  gc_DbmTranslation_en_Text2282 : WSTRING(21) := "Variable debug Neotec";
  gc_DbmTranslation_en_Text2283 : WSTRING(21) := "Variable debug Neotec";
  gc_DbmTranslation_en_Text2284 : WSTRING(21) := "Variable debug Neotec";
  gc_DbmTranslation_en_Text2285 : WSTRING(21) := "Variable debug Neotec";
  gc_DbmTranslation_en_Text2286 : WSTRING(21) := "Variable debug Neotec";
  gc_DbmTranslation_en_Text2287 : WSTRING(21) := "Variable debug Neotec";
  gc_DbmTranslation_en_Text2288 : WSTRING(21) := "Variable debug Neotec";
  gc_DbmTranslation_en_Text2289 : WSTRING(21) := "Variable debug Neotec";
  gc_DbmTranslation_en_Text2290 : WSTRING(21) := "Variable debug Neotec";
  gc_DbmTranslation_en_Text2291 : WSTRING(21) := "Variable debug Neotec";
  gc_DbmTranslation_en_Text2292 : WSTRING(21) := "Variable debug Neotec";
  gc_DbmTranslation_en_Text2293 : WSTRING(21) := "Variable debug Neotec";
  gc_DbmTranslation_en_Text2294 : WSTRING(21) := "Variable debug Neotec";
  gc_DbmTranslation_en_Text2295 : WSTRING(21) := "Variable debug Neotec";
  gc_DbmTranslation_en_Text2296 : WSTRING(21) := "Variable debug Neotec";
  gc_DbmTranslation_en_Text2297 : WSTRING(21) := "Variable debug Neotec";
  gc_DbmTranslation_en_Text2298 : WSTRING(21) := "Variable debug Neotec";
  gc_DbmTranslation_en_Text2299 : WSTRING(21) := "Variable debug Neotec";
  gc_DbmTranslation_en_Text2300 : WSTRING(21) := "Variable debug Neotec";
  gc_DbmTranslation_en_Text2301 : WSTRING(21) := "Variable debug Neotec";
  gc_DbmTranslation_en_Text2302 : WSTRING(21) := "Variable debug Neotec";
  gc_DbmTranslation_en_Text2303 : WSTRING(21) := "Variable debug Neotec";
  gc_DbmTranslation_en_Text2304 : WSTRING(21) := "Variable debug Neotec";
  gc_DbmTranslation_en_Text2305 : WSTRING(21) := "Variable debug Neotec";
  gc_DbmTranslation_en_Text2306 : WSTRING(21) := "Variable debug Neotec";
  gc_DbmTranslation_en_Text2307 : WSTRING(21) := "Variable debug Neotec";
  gc_DbmTranslation_en_Text2308 : WSTRING(21) := "Variable debug Neotec";
  gc_DbmTranslation_en_Text2309 : WSTRING(21) := "Variable debug Neotec";
  gc_DbmTranslation_en_Text2310 : WSTRING(21) := "Variable debug Neotec";
  gc_DbmTranslation_en_Text2311 : WSTRING(64) := "Mesure de la température du liquide de refroidissement du moteur";
  gc_DbmTranslation_en_Text2312 : WSTRING(58) := "Pression mesuré dans le système de lubrification du moteur";
  gc_DbmTranslation_en_Text2313 : WSTRING(34) := "Vitesse actuelle du moteur calculé";
  gc_DbmTranslation_en_Text2314 : WSTRING(56) := "Courant de l'alternateur principale du moteur thermique ";
  gc_DbmTranslation_en_Text2315 : WSTRING(56) := "Etat du moteur : Motor stop, pre-start, Wram-Up,Starting";
  gc_DbmTranslation_en_Text2316 : WSTRING(40) := "Tension mesuré aux bornes de la batterie";
  gc_DbmTranslation_en_Text2317 : WSTRING(33) := "Commande de la vietesse du moteur";
  gc_DbmTranslation_en_Text2318 : WSTRING(30) := "Override Control Mode (SPN695)";
  gc_DbmTranslation_en_Text2319 : WSTRING(18) := "High pressure Oil ";
  gc_DbmTranslation_en_Text2320 : WSTRING(14) := "Warmin gActive";
  gc_DbmTranslation_en_Text2321 : WSTRING(10) := "Stop Motor";
  gc_DbmTranslation_en_Text2322 : WSTRING(27) := "Regeneration SOC at maximum";
  gc_DbmTranslation_en_Text2323 : WSTRING(61) := "Threshold maximum to autorize regeneration (Threshold of SOC)";
  gc_DbmTranslation_en_Text2324 : WSTRING(42) := "Hysteresis for regeneration of SOC maximum";
  gc_DbmTranslation_en_Text2325 : WSTRING(57) := "Number of time to refuse reloading from generator (Alarm)";
  gc_DbmTranslation_en_Text2326 : WSTRING(61) := "Number of time to refuse reloading from generator (forbidden)";
  gc_DbmTranslation_en_Text2327 : WSTRING(23) := "RPM motor maximum value";
  gc_DbmTranslation_en_Text2328 : WSTRING(23) := "RPM motor minimum value";
  gc_DbmTranslation_en_Text2329 : WSTRING(27) := "RPM for a movement with PVG";
  gc_DbmTranslation_en_Text2330 : WSTRING(27) := "RPM for a movement with TOR";
  gc_DbmTranslation_en_Text2331 : WSTRING(30) := "Hydraulic oil cold temperature";
  gc_DbmTranslation_en_Text2332 : WSTRING(42) := "Capacity of the battery in ampere per hour";
  gc_DbmTranslation_en_Text2333 : WSTRING(53) := "Number of element for the remaining regeneration time";
  gc_DbmTranslation_en_Text2334 : WSTRING(61) := "Number of times the alarm regeneration threshold was exceeded";
  gc_DbmTranslation_en_Text2335 : WSTRING(89) := "Number of times we exceeded the threshold of regeneration forbidden of the electric motor";
  gc_DbmTranslation_en_Text2336 : WSTRING(25) := "Cold Oil Tank Temperature";
  gc_DbmTranslation_en_Text2337 : WSTRING(30) := "Rpm Movements on Electric Mode";
  gc_DbmTranslation_en_Text2338 : WSTRING(37) := "Rpm Translation on Rail Electric Mode";
  gc_DbmTranslation_en_Text2339 : WSTRING(24) := "Rpm Oil Tank Temperature";
  gc_DbmTranslation_en_Text2340 : WSTRING(18) := "Rpm Electric motor";
  gc_DbmTranslation_en_Text2341 : WSTRING(12) := "Generator ON";
  gc_DbmTranslation_en_Text2342 : WSTRING(23) := "Automatic mode activate";
  gc_DbmTranslation_en_Text2343 : WSTRING(21) := "Silence mode activate";
  gc_DbmTranslation_en_Text2344 : WSTRING(21) := "Forcing mode activate";
  gc_DbmTranslation_en_Text2345 : WSTRING(24) := "Forcing regeneration Low";
  gc_DbmTranslation_en_Text2346 : WSTRING(25) := "Forcing regeneration High";
  gc_DbmTranslation_en_Text2347 : WSTRING(35) := "Remaining Regeneration time average";
  gc_DbmTranslation_en_Text2348 : WSTRING(25) := "Ask Reload With Generator";
  gc_DbmTranslation_en_Text2349 : WSTRING(27) := "Reloading With Generator On";
  gc_DbmTranslation_en_Text2350 : WSTRING(24) := "Stop regeneration by SOC";
  gc_DbmTranslation_en_Text2351 : WSTRING(24) := "Total regeneration Hours";
  gc_DbmTranslation_en_Text2352 : WSTRING(31) := "Picto Cold Oil Tank Temperature";
  gc_DbmTranslation_en_Text2353 : WSTRING(20) := "Total electric hours";
  gc_DbmTranslation_en_Text2354 : WSTRING(37) := "Picto recovery reduction ratio active";
  gc_DbVarGrpNameTranslation_en_Text2355 : WSTRING(17) := "NV_PARAMERTERS_C0";
  gc_DbVarGrpNameTranslation_en_Text2356 : WSTRING(23) := "NV_PARAM_SPEED_MAX_RAIL";
  gc_DbVarGrpNameTranslation_en_Text2357 : WSTRING(19) := "NV_PARAM_BRAKE_TEST";
  gc_DbVarGrpNameTranslation_en_Text2358 : WSTRING(28) := "NV_PARAM_RAIL_WORK_SAFETY_C0";
  gc_DbVarGrpNameTranslation_en_Text2359 : WSTRING(25) := "NV_PARAM_TRANSPORT_POS_C0";
  gc_DbVarGrpNameTranslation_en_Text2360 : WSTRING(28) := "NV_PARAM_SELECT_CONTROL_POST";
  gc_DbVarGrpNameTranslation_en_Text2361 : WSTRING(17) := "NV_PARAM_ALARM_C0";
  gc_DbVarGrpNameTranslation_en_Text2362 : WSTRING(21) := "NV_PARAM_MAST_DISPLAY";
  gc_DbVarGrpNameTranslation_en_Text2363 : WSTRING(17) := "NV_PARAMERTERS_C1";
  gc_DbVarGrpNameTranslation_en_Text2364 : WSTRING(17) := "NV_PARAM_MOTOR_C1";
  gc_DbVarGrpNameTranslation_en_Text2365 : WSTRING(31) := "NV_PARAM_LIMIT_WORK_ENVELOPE_C1";
  gc_DbVarGrpNameTranslation_en_Text2366 : WSTRING(24) := "NV_PARAM_MVT_END_STOP_C1";
  gc_DbVarGrpNameTranslation_en_Text2367 : WSTRING(21) := "NV_PARAM_AUTO_STOP_C1";
  gc_DbVarGrpNameTranslation_en_Text2368 : WSTRING(16) := "NV_PARAM_MAST_C1";
  gc_DbVarGrpNameTranslation_en_Text2369 : WSTRING(17) := "NV_PARAM_ALARM_C1";
  gc_DbVarGrpNameTranslation_en_Text2370 : WSTRING(12) := "NV_OPTION_C0";
  gc_DbVarGrpNameTranslation_en_Text2371 : WSTRING(12) := "NV_OPTION_C1";
  gc_DbmTranslation_en_Texts : ARRAY[0..2371] OF POINTER TO WSTRING(123) := [ADR(gc_DbmTranslation_en_Text0), ADR(gc_DbmTranslation_en_Text1), ADR(gc_DbmTranslation_en_Text2), ADR(gc_DbmTranslation_en_Text3), ADR(gc_DbmTranslation_en_Text4), ADR(gc_DbmTranslation_en_Text5), ADR(gc_DbmTranslation_en_Text6), ADR(gc_DbmTranslation_en_Text7), ADR(gc_DbmTranslation_en_Text8), ADR(gc_DbmTranslation_en_Text9), ADR(gc_DbmTranslation_en_Text10), ADR(gc_DbmTranslation_en_Text11), ADR(gc_DbmTranslation_en_Text12), ADR(gc_DbmTranslation_en_Text13), ADR(gc_DbmTranslation_en_Text14), ADR(gc_DbmTranslation_en_Text15), ADR(gc_DbmTranslation_en_Text16), ADR(gc_DbmTranslation_en_Text17), ADR(gc_DbmTranslation_en_Text18), ADR(gc_DbmTranslation_en_Text19), ADR(gc_DbmTranslation_en_Text20), ADR(gc_DbmTranslation_en_Text21), ADR(gc_DbmTranslation_en_Text22), ADR(gc_DbmTranslation_en_Text23), ADR(gc_DbmTranslation_en_Text24), ADR(gc_DbmTranslation_en_Text25), ADR(gc_DbmTranslation_en_Text26), ADR(gc_DbmTranslation_en_Text27), ADR(gc_DbmTranslation_en_Text28), ADR(gc_DbmTranslation_en_Text29), ADR(gc_DbmTranslation_en_Text30), ADR(gc_DbmTranslation_en_Text31), ADR(gc_DbmTranslation_en_Text32), ADR(gc_DbmTranslation_en_Text33), ADR(gc_DbmTranslation_en_Text34), ADR(gc_DbmTranslation_en_Text35), ADR(gc_DbmTranslation_en_Text36), ADR(gc_DbmTranslation_en_Text37), ADR(gc_DbmTranslation_en_Text38), ADR(gc_DbmTranslation_en_Text39), ADR(gc_DbmTranslation_en_Text40), ADR(gc_DbmTranslation_en_Text41), ADR(gc_DbmTranslation_en_Text42), ADR(gc_DbmTranslation_en_Text43), ADR(gc_DbmTranslation_en_Text44), ADR(gc_DbmTranslation_en_Text45), ADR(gc_DbmTranslation_en_Text46), ADR(gc_DbmTranslation_en_Text47), ADR(gc_DbmTranslation_en_Text48), ADR(gc_DbmTranslation_en_Text49), ADR(gc_DbmTranslation_en_Text50), ADR(gc_DbmTranslation_en_Text51), ADR(gc_DbmTranslation_en_Text52), ADR(gc_DbmTranslation_en_Text53), ADR(gc_DbmTranslation_en_Text54), ADR(gc_DbmTranslation_en_Text55), ADR(gc_DbmTranslation_en_Text56), ADR(gc_DbmTranslation_en_Text57), ADR(gc_DbmTranslation_en_Text58), ADR(gc_DbmTranslation_en_Text59), ADR(gc_DbmTranslation_en_Text60), ADR(gc_DbmTranslation_en_Text61), ADR(gc_DbmTranslation_en_Text62), ADR(gc_DbmTranslation_en_Text63), ADR(gc_DbmTranslation_en_Text64), ADR(gc_DbmTranslation_en_Text65), ADR(gc_DbmTranslation_en_Text66), ADR(gc_DbmTranslation_en_Text67), ADR(gc_DbmTranslation_en_Text68), ADR(gc_DbmTranslation_en_Text69), ADR(gc_DbmTranslation_en_Text70), ADR(gc_DbmTranslation_en_Text71), ADR(gc_DbmTranslation_en_Text72), ADR(gc_DbmTranslation_en_Text73), ADR(gc_DbmTranslation_en_Text74), ADR(gc_DbmTranslation_en_Text75), ADR(gc_DbmTranslation_en_Text76), ADR(gc_DbmTranslation_en_Text77), ADR(gc_DbmTranslation_en_Text78), ADR(gc_DbmTranslation_en_Text79), ADR(gc_DbmTranslation_en_Text80), ADR(gc_DbmTranslation_en_Text81), ADR(gc_DbmTranslation_en_Text82), ADR(gc_DbmTranslation_en_Text83), ADR(gc_DbmTranslation_en_Text84), ADR(gc_DbmTranslation_en_Text85), ADR(gc_DbmTranslation_en_Text86), ADR(gc_DbmTranslation_en_Text87), ADR(gc_DbmTranslation_en_Text88), ADR(gc_DbmTranslation_en_Text89), ADR(gc_DbmTranslation_en_Text90), ADR(gc_DbmTranslation_en_Text91), ADR(gc_DbmTranslation_en_Text92), ADR(gc_DbmTranslation_en_Text93), ADR(gc_DbmTranslation_en_Text94), ADR(gc_DbmTranslation_en_Text95), ADR(gc_DbmTranslation_en_Text96), ADR(gc_DbmTranslation_en_Text97), ADR(gc_DbmTranslation_en_Text98), ADR(gc_DbmTranslation_en_Text99), ADR(gc_DbmTranslation_en_Text100), ADR(gc_DbmTranslation_en_Text101), ADR(gc_DbmTranslation_en_Text102), ADR(gc_DbmTranslation_en_Text103), ADR(gc_DbmTranslation_en_Text104), ADR(gc_DbmTranslation_en_Text105), ADR(gc_DbmTranslation_en_Text106), ADR(gc_DbmTranslation_en_Text107), ADR(gc_DbmTranslation_en_Text108), ADR(gc_DbmTranslation_en_Text109), ADR(gc_DbmTranslation_en_Text110), ADR(gc_DbmTranslation_en_Text111), ADR(gc_DbmTranslation_en_Text112), ADR(gc_DbmTranslation_en_Text113), ADR(gc_DbmTranslation_en_Text114), ADR(gc_DbmTranslation_en_Text115), ADR(gc_DbmTranslation_en_Text116), ADR(gc_DbmTranslation_en_Text117), ADR(gc_DbmTranslation_en_Text118), ADR(gc_DbmTranslation_en_Text119), ADR(gc_DbmTranslation_en_Text120), ADR(gc_DbmTranslation_en_Text121), ADR(gc_DbmTranslation_en_Text122), ADR(gc_DbmTranslation_en_Text123), ADR(gc_DbmTranslation_en_Text124), ADR(gc_DbmTranslation_en_Text125), ADR(gc_DbmTranslation_en_Text126), ADR(gc_DbmTranslation_en_Text127), ADR(gc_DbmTranslation_en_Text128), ADR(gc_DbmTranslation_en_Text129), ADR(gc_DbmTranslation_en_Text130), ADR(gc_DbmTranslation_en_Text131), ADR(gc_DbmTranslation_en_Text132), ADR(gc_DbmTranslation_en_Text133), ADR(gc_DbmTranslation_en_Text134), ADR(gc_DbmTranslation_en_Text135), ADR(gc_DbmTranslation_en_Text136), ADR(gc_DbmTranslation_en_Text137), ADR(gc_DbmTranslation_en_Text138), ADR(gc_DbmTranslation_en_Text139), ADR(gc_DbmTranslation_en_Text140), ADR(gc_DbmTranslation_en_Text141), ADR(gc_DbmTranslation_en_Text142), ADR(gc_DbmTranslation_en_Text143), ADR(gc_DbmTranslation_en_Text144), ADR(gc_DbmTranslation_en_Text145), ADR(gc_DbmTranslation_en_Text146), ADR(gc_DbmTranslation_en_Text147), ADR(gc_DbmTranslation_en_Text148), ADR(gc_DbmTranslation_en_Text149), ADR(gc_DbmTranslation_en_Text150), ADR(gc_DbmTranslation_en_Text151), ADR(gc_DbmTranslation_en_Text152), ADR(gc_DbmTranslation_en_Text153), ADR(gc_DbmTranslation_en_Text154), ADR(gc_DbmTranslation_en_Text155), ADR(gc_DbmTranslation_en_Text156), ADR(gc_DbmTranslation_en_Text157), ADR(gc_DbmTranslation_en_Text158), ADR(gc_DbmTranslation_en_Text159), ADR(gc_DbmTranslation_en_Text160), ADR(gc_DbmTranslation_en_Text161), ADR(gc_DbmTranslation_en_Text162), ADR(gc_DbmTranslation_en_Text163), ADR(gc_DbmTranslation_en_Text164), ADR(gc_DbmTranslation_en_Text165), ADR(gc_DbmTranslation_en_Text166), ADR(gc_DbmTranslation_en_Text167), ADR(gc_DbmTranslation_en_Text168), ADR(gc_DbmTranslation_en_Text169), ADR(gc_DbmTranslation_en_Text170), ADR(gc_DbmTranslation_en_Text171), ADR(gc_DbmTranslation_en_Text172), ADR(gc_DbmTranslation_en_Text173), ADR(gc_DbmTranslation_en_Text174), ADR(gc_DbmTranslation_en_Text175), ADR(gc_DbmTranslation_en_Text176), ADR(gc_DbmTranslation_en_Text177), ADR(gc_DbmTranslation_en_Text178), ADR(gc_DbmTranslation_en_Text179), ADR(gc_DbmTranslation_en_Text180), ADR(gc_DbmTranslation_en_Text181), ADR(gc_DbmTranslation_en_Text182), ADR(gc_DbmTranslation_en_Text183), ADR(gc_DbmTranslation_en_Text184), ADR(gc_DbmTranslation_en_Text185), ADR(gc_DbmTranslation_en_Text186), ADR(gc_DbmTranslation_en_Text187), ADR(gc_DbmTranslation_en_Text188), ADR(gc_DbmTranslation_en_Text189), ADR(gc_DbmTranslation_en_Text190), ADR(gc_DbmTranslation_en_Text191), ADR(gc_DbmTranslation_en_Text192), ADR(gc_DbmTranslation_en_Text193), ADR(gc_DbmTranslation_en_Text194), ADR(gc_DbmTranslation_en_Text195), ADR(gc_DbmTranslation_en_Text196), ADR(gc_DbmTranslation_en_Text197), ADR(gc_DbmTranslation_en_Text198), ADR(gc_DbmTranslation_en_Text199), ADR(gc_DbmTranslation_en_Text200), ADR(gc_DbmTranslation_en_Text201), ADR(gc_DbmTranslation_en_Text202), ADR(gc_DbmTranslation_en_Text203), ADR(gc_DbmTranslation_en_Text204), ADR(gc_DbmTranslation_en_Text205), ADR(gc_DbmTranslation_en_Text206), ADR(gc_DbmTranslation_en_Text207), ADR(gc_DbmTranslation_en_Text208), ADR(gc_DbmTranslation_en_Text209), ADR(gc_DbmTranslation_en_Text210), ADR(gc_DbmTranslation_en_Text211), ADR(gc_DbmTranslation_en_Text212), ADR(gc_DbmTranslation_en_Text213), ADR(gc_DbmTranslation_en_Text214), ADR(gc_DbmTranslation_en_Text215), ADR(gc_DbmTranslation_en_Text216), ADR(gc_DbmTranslation_en_Text217), ADR(gc_DbmTranslation_en_Text218), ADR(gc_DbmTranslation_en_Text219), ADR(gc_DbmTranslation_en_Text220), ADR(gc_DbmTranslation_en_Text221), ADR(gc_DbmTranslation_en_Text222), ADR(gc_DbmTranslation_en_Text223), ADR(gc_DbmTranslation_en_Text224), ADR(gc_DbmTranslation_en_Text225), ADR(gc_DbmTranslation_en_Text226), ADR(gc_DbmTranslation_en_Text227), ADR(gc_DbmTranslation_en_Text228), ADR(gc_DbmTranslation_en_Text229), ADR(gc_DbmTranslation_en_Text230), ADR(gc_DbmTranslation_en_Text231), ADR(gc_DbmTranslation_en_Text232), ADR(gc_DbmTranslation_en_Text233), ADR(gc_DbmTranslation_en_Text234), ADR(gc_DbmTranslation_en_Text235), ADR(gc_DbmTranslation_en_Text236), ADR(gc_DbmTranslation_en_Text237), ADR(gc_DbmTranslation_en_Text238), ADR(gc_DbmTranslation_en_Text239), ADR(gc_DbmTranslation_en_Text240), ADR(gc_DbmTranslation_en_Text241), ADR(gc_DbmTranslation_en_Text242), ADR(gc_DbmTranslation_en_Text243), ADR(gc_DbmTranslation_en_Text244), ADR(gc_DbmTranslation_en_Text245), ADR(gc_DbmTranslation_en_Text246), ADR(gc_DbmTranslation_en_Text247), ADR(gc_DbmTranslation_en_Text248), ADR(gc_DbmTranslation_en_Text249), ADR(gc_DbmTranslation_en_Text250), ADR(gc_DbmTranslation_en_Text251), ADR(gc_DbmTranslation_en_Text252), ADR(gc_DbmTranslation_en_Text253), ADR(gc_DbmTranslation_en_Text254), ADR(gc_DbmTranslation_en_Text255), ADR(gc_DbmTranslation_en_Text256), ADR(gc_DbmTranslation_en_Text257), ADR(gc_DbmTranslation_en_Text258), ADR(gc_DbmTranslation_en_Text259), ADR(gc_DbmTranslation_en_Text260), ADR(gc_DbmTranslation_en_Text261), ADR(gc_DbmTranslation_en_Text262), ADR(gc_DbmTranslation_en_Text263), ADR(gc_DbmTranslation_en_Text264), ADR(gc_DbmTranslation_en_Text265), ADR(gc_DbmTranslation_en_Text266), ADR(gc_DbmTranslation_en_Text267), ADR(gc_DbmTranslation_en_Text268), ADR(gc_DbmTranslation_en_Text269), ADR(gc_DbmTranslation_en_Text270), ADR(gc_DbmTranslation_en_Text271), ADR(gc_DbmTranslation_en_Text272), ADR(gc_DbmTranslation_en_Text273), ADR(gc_DbmTranslation_en_Text274), ADR(gc_DbmTranslation_en_Text275), ADR(gc_DbmTranslation_en_Text276), ADR(gc_DbmTranslation_en_Text277), ADR(gc_DbmTranslation_en_Text278), ADR(gc_DbmTranslation_en_Text279), ADR(gc_DbmTranslation_en_Text280), ADR(gc_DbmTranslation_en_Text281), ADR(gc_DbmTranslation_en_Text282), ADR(gc_DbmTranslation_en_Text283), ADR(gc_DbmTranslation_en_Text284), ADR(gc_DbmTranslation_en_Text285), ADR(gc_DbmTranslation_en_Text286), ADR(gc_DbmTranslation_en_Text287), ADR(gc_DbmTranslation_en_Text288), ADR(gc_DbmTranslation_en_Text289), ADR(gc_DbmTranslation_en_Text290), ADR(gc_DbmTranslation_en_Text291), ADR(gc_DbmTranslation_en_Text292), ADR(gc_DbmTranslation_en_Text293), ADR(gc_DbmTranslation_en_Text294), ADR(gc_DbmTranslation_en_Text295), ADR(gc_DbmTranslation_en_Text296), ADR(gc_DbmTranslation_en_Text297), ADR(gc_DbmTranslation_en_Text298), ADR(gc_DbmTranslation_en_Text299), ADR(gc_DbmTranslation_en_Text300), ADR(gc_DbmTranslation_en_Text301), ADR(gc_DbmTranslation_en_Text302), ADR(gc_DbmTranslation_en_Text303), ADR(gc_DbmTranslation_en_Text304), ADR(gc_DbmTranslation_en_Text305), ADR(gc_DbmTranslation_en_Text306), ADR(gc_DbmTranslation_en_Text307), ADR(gc_DbmTranslation_en_Text308), ADR(gc_DbmTranslation_en_Text309), ADR(gc_DbmTranslation_en_Text310), ADR(gc_DbmTranslation_en_Text311), ADR(gc_DbmTranslation_en_Text312), ADR(gc_DbmTranslation_en_Text313), ADR(gc_DbmTranslation_en_Text314), ADR(gc_DbmTranslation_en_Text315), ADR(gc_DbmTranslation_en_Text316), ADR(gc_DbmTranslation_en_Text317), ADR(gc_DbmTranslation_en_Text318), ADR(gc_DbmTranslation_en_Text319), ADR(gc_DbmTranslation_en_Text320), ADR(gc_DbmTranslation_en_Text321), ADR(gc_DbmTranslation_en_Text322), ADR(gc_DbmTranslation_en_Text323), ADR(gc_DbmTranslation_en_Text324), ADR(gc_DbmTranslation_en_Text325), ADR(gc_DbmTranslation_en_Text326), ADR(gc_DbmTranslation_en_Text327), ADR(gc_DbmTranslation_en_Text328), ADR(gc_DbmTranslation_en_Text329), ADR(gc_DbmTranslation_en_Text330), ADR(gc_DbmTranslation_en_Text331), ADR(gc_DbmTranslation_en_Text332), ADR(gc_DbmTranslation_en_Text333), ADR(gc_DbmTranslation_en_Text334), ADR(gc_DbmTranslation_en_Text335), ADR(gc_DbmTranslation_en_Text336), ADR(gc_DbmTranslation_en_Text337), ADR(gc_DbmTranslation_en_Text338), ADR(gc_DbmTranslation_en_Text339), ADR(gc_DbmTranslation_en_Text340), ADR(gc_DbmTranslation_en_Text341), ADR(gc_DbmTranslation_en_Text342), ADR(gc_DbmTranslation_en_Text343), ADR(gc_DbmTranslation_en_Text344), ADR(gc_DbmTranslation_en_Text345), ADR(gc_DbmTranslation_en_Text346), ADR(gc_DbmTranslation_en_Text347), ADR(gc_DbmTranslation_en_Text348), ADR(gc_DbmTranslation_en_Text349), ADR(gc_DbmTranslation_en_Text350), ADR(gc_DbmTranslation_en_Text351), ADR(gc_DbmTranslation_en_Text352), ADR(gc_DbmTranslation_en_Text353), ADR(gc_DbmTranslation_en_Text354), ADR(gc_DbmTranslation_en_Text355), ADR(gc_DbmTranslation_en_Text356), ADR(gc_DbmTranslation_en_Text357), ADR(gc_DbmTranslation_en_Text358), ADR(gc_DbmTranslation_en_Text359), ADR(gc_DbmTranslation_en_Text360), ADR(gc_DbmTranslation_en_Text361), ADR(gc_DbmTranslation_en_Text362), ADR(gc_DbmTranslation_en_Text363), ADR(gc_DbmTranslation_en_Text364), ADR(gc_DbmTranslation_en_Text365), ADR(gc_DbmTranslation_en_Text366), ADR(gc_DbmTranslation_en_Text367), ADR(gc_DbmTranslation_en_Text368), ADR(gc_DbmTranslation_en_Text369), ADR(gc_DbmTranslation_en_Text370), ADR(gc_DbmTranslation_en_Text371), ADR(gc_DbmTranslation_en_Text372), ADR(gc_DbmTranslation_en_Text373), ADR(gc_DbmTranslation_en_Text374), ADR(gc_DbmTranslation_en_Text375), ADR(gc_DbmTranslation_en_Text376), ADR(gc_DbmTranslation_en_Text377), ADR(gc_DbmTranslation_en_Text378), ADR(gc_DbmTranslation_en_Text379), ADR(gc_DbmTranslation_en_Text380), ADR(gc_DbmTranslation_en_Text381), ADR(gc_DbmTranslation_en_Text382), ADR(gc_DbmTranslation_en_Text383), ADR(gc_DbmTranslation_en_Text384), ADR(gc_DbmTranslation_en_Text385), ADR(gc_DbmTranslation_en_Text386), ADR(gc_DbmTranslation_en_Text387), ADR(gc_DbmTranslation_en_Text388), ADR(gc_DbmTranslation_en_Text389), ADR(gc_DbmTranslation_en_Text390), ADR(gc_DbmTranslation_en_Text391), ADR(gc_DbmTranslation_en_Text392), ADR(gc_DbmTranslation_en_Text393), ADR(gc_DbmTranslation_en_Text394), ADR(gc_DbmTranslation_en_Text395), ADR(gc_DbmTranslation_en_Text396), ADR(gc_DbmTranslation_en_Text397), ADR(gc_DbmTranslation_en_Text398), ADR(gc_DbmTranslation_en_Text399), ADR(gc_DbmTranslation_en_Text400), ADR(gc_DbmTranslation_en_Text401), ADR(gc_DbmTranslation_en_Text402), ADR(gc_DbmTranslation_en_Text403), ADR(gc_DbmTranslation_en_Text404), ADR(gc_DbmTranslation_en_Text405), ADR(gc_DbmTranslation_en_Text406), ADR(gc_DbmTranslation_en_Text407), ADR(gc_DbmTranslation_en_Text408), ADR(gc_DbmTranslation_en_Text409), ADR(gc_DbmTranslation_en_Text410), ADR(gc_DbmTranslation_en_Text411), ADR(gc_DbmTranslation_en_Text412), ADR(gc_DbmTranslation_en_Text413), ADR(gc_DbmTranslation_en_Text414), ADR(gc_DbmTranslation_en_Text415), ADR(gc_DbmTranslation_en_Text416), ADR(gc_DbmTranslation_en_Text417), ADR(gc_DbmTranslation_en_Text418), ADR(gc_DbmTranslation_en_Text419), ADR(gc_DbmTranslation_en_Text420), ADR(gc_DbmTranslation_en_Text421), ADR(gc_DbmTranslation_en_Text422), ADR(gc_DbmTranslation_en_Text423), ADR(gc_DbmTranslation_en_Text424), ADR(gc_DbmTranslation_en_Text425), ADR(gc_DbmTranslation_en_Text426), ADR(gc_DbmTranslation_en_Text427), ADR(gc_DbmTranslation_en_Text428), ADR(gc_DbmTranslation_en_Text429), ADR(gc_DbmTranslation_en_Text430), ADR(gc_DbmTranslation_en_Text431), ADR(gc_DbmTranslation_en_Text432), ADR(gc_DbmTranslation_en_Text433), ADR(gc_DbmTranslation_en_Text434), ADR(gc_DbmTranslation_en_Text435), ADR(gc_DbmTranslation_en_Text436), ADR(gc_DbmTranslation_en_Text437), ADR(gc_DbmTranslation_en_Text438), ADR(gc_DbmTranslation_en_Text439), ADR(gc_DbmTranslation_en_Text440), ADR(gc_DbmTranslation_en_Text441), ADR(gc_DbmTranslation_en_Text442), ADR(gc_DbmTranslation_en_Text443), ADR(gc_DbmTranslation_en_Text444), ADR(gc_DbmTranslation_en_Text445), ADR(gc_DbmTranslation_en_Text446), ADR(gc_DbmTranslation_en_Text447), ADR(gc_DbmTranslation_en_Text448), ADR(gc_DbmTranslation_en_Text449), ADR(gc_DbmTranslation_en_Text450), ADR(gc_DbmTranslation_en_Text451), ADR(gc_DbmTranslation_en_Text452), ADR(gc_DbmTranslation_en_Text453), ADR(gc_DbmTranslation_en_Text454), ADR(gc_DbmTranslation_en_Text455), ADR(gc_DbmTranslation_en_Text456), ADR(gc_DbmTranslation_en_Text457), ADR(gc_DbmTranslation_en_Text458), ADR(gc_DbmTranslation_en_Text459), ADR(gc_DbmTranslation_en_Text460), ADR(gc_DbmTranslation_en_Text461), ADR(gc_DbmTranslation_en_Text462), ADR(gc_DbmTranslation_en_Text463), ADR(gc_DbmTranslation_en_Text464), ADR(gc_DbmTranslation_en_Text465), ADR(gc_DbmTranslation_en_Text466), ADR(gc_DbmTranslation_en_Text467), ADR(gc_DbmTranslation_en_Text468), ADR(gc_DbmTranslation_en_Text469), ADR(gc_DbmTranslation_en_Text470), ADR(gc_DbmTranslation_en_Text471), ADR(gc_DbmTranslation_en_Text472), ADR(gc_DbmTranslation_en_Text473), ADR(gc_DbmTranslation_en_Text474), ADR(gc_DbmTranslation_en_Text475), ADR(gc_DbmTranslation_en_Text476), ADR(gc_DbmTranslation_en_Text477), ADR(gc_DbmTranslation_en_Text478), ADR(gc_DbmTranslation_en_Text479), ADR(gc_DbmTranslation_en_Text480), ADR(gc_DbmTranslation_en_Text481), ADR(gc_DbmTranslation_en_Text482), ADR(gc_DbmTranslation_en_Text483), ADR(gc_DbmTranslation_en_Text484), ADR(gc_DbmTranslation_en_Text485), ADR(gc_DbmTranslation_en_Text486), ADR(gc_DbmTranslation_en_Text487), ADR(gc_DbmTranslation_en_Text488), ADR(gc_DbmTranslation_en_Text489), ADR(gc_DbmTranslation_en_Text490), ADR(gc_DbmTranslation_en_Text491), ADR(gc_DbmTranslation_en_Text492), ADR(gc_DbmTranslation_en_Text493), ADR(gc_DbmTranslation_en_Text494), ADR(gc_DbmTranslation_en_Text495), ADR(gc_DbmTranslation_en_Text496), ADR(gc_DbmTranslation_en_Text497), ADR(gc_DbmTranslation_en_Text498), ADR(gc_DbmTranslation_en_Text499), ADR(gc_DbmTranslation_en_Text500), ADR(gc_DbmTranslation_en_Text501), ADR(gc_DbmTranslation_en_Text502), ADR(gc_DbmTranslation_en_Text503), ADR(gc_DbmTranslation_en_Text504), ADR(gc_DbmTranslation_en_Text505), ADR(gc_DbmTranslation_en_Text506), ADR(gc_DbmTranslation_en_Text507), ADR(gc_DbmTranslation_en_Text508), ADR(gc_DbmTranslation_en_Text509), ADR(gc_DbmTranslation_en_Text510), ADR(gc_DbmTranslation_en_Text511), ADR(gc_DbmTranslation_en_Text512), ADR(gc_DbmTranslation_en_Text513), ADR(gc_DbmTranslation_en_Text514), ADR(gc_DbmTranslation_en_Text515), ADR(gc_DbmTranslation_en_Text516), ADR(gc_DbmTranslation_en_Text517), ADR(gc_DbmTranslation_en_Text518), ADR(gc_DbmTranslation_en_Text519), ADR(gc_DbmTranslation_en_Text520), ADR(gc_DbmTranslation_en_Text521), ADR(gc_DbmTranslation_en_Text522), ADR(gc_DbmTranslation_en_Text523), ADR(gc_DbmTranslation_en_Text524), ADR(gc_DbmTranslation_en_Text525), ADR(gc_DbmTranslation_en_Text526), ADR(gc_DbmTranslation_en_Text527), ADR(gc_DbmTranslation_en_Text528), ADR(gc_DbmTranslation_en_Text529), ADR(gc_DbmTranslation_en_Text530), ADR(gc_DbmTranslation_en_Text531), ADR(gc_DbmTranslation_en_Text532), ADR(gc_DbmTranslation_en_Text533), ADR(gc_DbmTranslation_en_Text534), ADR(gc_DbmTranslation_en_Text535), ADR(gc_DbmTranslation_en_Text536), ADR(gc_DbmTranslation_en_Text537), ADR(gc_DbmTranslation_en_Text538), ADR(gc_DbmTranslation_en_Text539), ADR(gc_DbmTranslation_en_Text540), ADR(gc_DbmTranslation_en_Text541), ADR(gc_DbmTranslation_en_Text542), ADR(gc_DbmTranslation_en_Text543), ADR(gc_DbmTranslation_en_Text544), ADR(gc_DbmTranslation_en_Text545), ADR(gc_DbmTranslation_en_Text546), ADR(gc_DbmTranslation_en_Text547), ADR(gc_DbmTranslation_en_Text548), ADR(gc_DbmTranslation_en_Text549), ADR(gc_DbmTranslation_en_Text550), ADR(gc_DbmTranslation_en_Text551), ADR(gc_DbmTranslation_en_Text552), ADR(gc_DbmTranslation_en_Text553), ADR(gc_DbmTranslation_en_Text554), ADR(gc_DbmTranslation_en_Text555), ADR(gc_DbmTranslation_en_Text556), ADR(gc_DbmTranslation_en_Text557), ADR(gc_DbmTranslation_en_Text558), ADR(gc_DbmTranslation_en_Text559), ADR(gc_DbmTranslation_en_Text560), ADR(gc_DbmTranslation_en_Text561), ADR(gc_DbmTranslation_en_Text562), ADR(gc_DbmTranslation_en_Text563), ADR(gc_DbmTranslation_en_Text564), ADR(gc_DbmTranslation_en_Text565), ADR(gc_DbmTranslation_en_Text566), ADR(gc_DbmTranslation_en_Text567), ADR(gc_DbmTranslation_en_Text568), ADR(gc_DbmTranslation_en_Text569), ADR(gc_DbmTranslation_en_Text570), ADR(gc_DbmTranslation_en_Text571), ADR(gc_DbmTranslation_en_Text572), ADR(gc_DbmTranslation_en_Text573), ADR(gc_DbmTranslation_en_Text574), ADR(gc_DbmTranslation_en_Text575), ADR(gc_DbmTranslation_en_Text576), ADR(gc_DbmTranslation_en_Text577), ADR(gc_DbmTranslation_en_Text578), ADR(gc_DbmTranslation_en_Text579), ADR(gc_DbmTranslation_en_Text580), ADR(gc_DbmTranslation_en_Text581), ADR(gc_DbmTranslation_en_Text582), ADR(gc_DbmTranslation_en_Text583), ADR(gc_DbmTranslation_en_Text584), ADR(gc_DbmTranslation_en_Text585), ADR(gc_DbmTranslation_en_Text586), ADR(gc_DbmTranslation_en_Text587), ADR(gc_DbmTranslation_en_Text588), ADR(gc_DbmTranslation_en_Text589), ADR(gc_DbmTranslation_en_Text590), ADR(gc_DbmTranslation_en_Text591), ADR(gc_DbmTranslation_en_Text592), ADR(gc_DbmTranslation_en_Text593), ADR(gc_DbmTranslation_en_Text594), ADR(gc_DbmTranslation_en_Text595), ADR(gc_DbmTranslation_en_Text596), ADR(gc_DbmTranslation_en_Text597), ADR(gc_DbmTranslation_en_Text598), ADR(gc_DbmTranslation_en_Text599), ADR(gc_DbmTranslation_en_Text600), ADR(gc_DbmTranslation_en_Text601), ADR(gc_DbmTranslation_en_Text602), ADR(gc_DbmTranslation_en_Text603), ADR(gc_DbmTranslation_en_Text604), ADR(gc_DbmTranslation_en_Text605), ADR(gc_DbmTranslation_en_Text606), ADR(gc_DbmTranslation_en_Text607), ADR(gc_DbmTranslation_en_Text608), ADR(gc_DbmTranslation_en_Text609), ADR(gc_DbmTranslation_en_Text610), ADR(gc_DbmTranslation_en_Text611), ADR(gc_DbmTranslation_en_Text612), ADR(gc_DbmTranslation_en_Text613), ADR(gc_DbmTranslation_en_Text614), ADR(gc_DbmTranslation_en_Text615), ADR(gc_DbmTranslation_en_Text616), ADR(gc_DbmTranslation_en_Text617), ADR(gc_DbmTranslation_en_Text618), ADR(gc_DbmTranslation_en_Text619), ADR(gc_DbmTranslation_en_Text620), ADR(gc_DbmTranslation_en_Text621), ADR(gc_DbmTranslation_en_Text622), ADR(gc_DbmTranslation_en_Text623), ADR(gc_DbmTranslation_en_Text624), ADR(gc_DbmTranslation_en_Text625), ADR(gc_DbmTranslation_en_Text626), ADR(gc_DbmTranslation_en_Text627), ADR(gc_DbmTranslation_en_Text628), ADR(gc_DbmTranslation_en_Text629), ADR(gc_DbmTranslation_en_Text630), ADR(gc_DbmTranslation_en_Text631), ADR(gc_DbmTranslation_en_Text632), ADR(gc_DbmTranslation_en_Text633), ADR(gc_DbmTranslation_en_Text634), ADR(gc_DbmTranslation_en_Text635), ADR(gc_DbmTranslation_en_Text636), ADR(gc_DbmTranslation_en_Text637), ADR(gc_DbmTranslation_en_Text638), ADR(gc_DbmTranslation_en_Text639), ADR(gc_DbmTranslation_en_Text640), ADR(gc_DbmTranslation_en_Text641), ADR(gc_DbmTranslation_en_Text642), ADR(gc_DbmTranslation_en_Text643), ADR(gc_DbmTranslation_en_Text644), ADR(gc_DbmTranslation_en_Text645), ADR(gc_DbmTranslation_en_Text646), ADR(gc_DbmTranslation_en_Text647), ADR(gc_DbmTranslation_en_Text648), ADR(gc_DbmTranslation_en_Text649), ADR(gc_DbmTranslation_en_Text650), ADR(gc_DbmTranslation_en_Text651), ADR(gc_DbmTranslation_en_Text652), ADR(gc_DbmTranslation_en_Text653), ADR(gc_DbmTranslation_en_Text654), ADR(gc_DbmTranslation_en_Text655), ADR(gc_DbmTranslation_en_Text656), ADR(gc_DbmTranslation_en_Text657), ADR(gc_DbmTranslation_en_Text658), ADR(gc_DbmTranslation_en_Text659), ADR(gc_DbmTranslation_en_Text660), ADR(gc_DbmTranslation_en_Text661), ADR(gc_DbmTranslation_en_Text662), ADR(gc_DbmTranslation_en_Text663), ADR(gc_DbmTranslation_en_Text664), ADR(gc_DbmTranslation_en_Text665), ADR(gc_DbmTranslation_en_Text666), ADR(gc_DbmTranslation_en_Text667), ADR(gc_DbmTranslation_en_Text668), ADR(gc_DbmTranslation_en_Text669), ADR(gc_DbmTranslation_en_Text670), ADR(gc_DbmTranslation_en_Text671), ADR(gc_DbmTranslation_en_Text672), ADR(gc_DbmTranslation_en_Text673), ADR(gc_DbmTranslation_en_Text674), ADR(gc_DbmTranslation_en_Text675), ADR(gc_DbmTranslation_en_Text676), ADR(gc_DbmTranslation_en_Text677), ADR(gc_DbmTranslation_en_Text678), ADR(gc_DbmTranslation_en_Text679), ADR(gc_DbmTranslation_en_Text680), ADR(gc_DbmTranslation_en_Text681), ADR(gc_DbmTranslation_en_Text682), ADR(gc_DbmTranslation_en_Text683), ADR(gc_DbmTranslation_en_Text684), ADR(gc_DbmTranslation_en_Text685), ADR(gc_DbmTranslation_en_Text686), ADR(gc_DbmTranslation_en_Text687), ADR(gc_DbmTranslation_en_Text688), ADR(gc_DbmTranslation_en_Text689), ADR(gc_DbmTranslation_en_Text690), ADR(gc_DbmTranslation_en_Text691), ADR(gc_DbmTranslation_en_Text692), ADR(gc_DbmTranslation_en_Text693), ADR(gc_DbmTranslation_en_Text694), ADR(gc_DbmTranslation_en_Text695), ADR(gc_DbmTranslation_en_Text696), ADR(gc_DbmTranslation_en_Text697), ADR(gc_DbmTranslation_en_Text698), ADR(gc_DbmTranslation_en_Text699), ADR(gc_DbmTranslation_en_Text700), ADR(gc_DbmTranslation_en_Text701), ADR(gc_DbmTranslation_en_Text702), ADR(gc_DbmTranslation_en_Text703), ADR(gc_DbmTranslation_en_Text704), ADR(gc_DbmTranslation_en_Text705), ADR(gc_DbmTranslation_en_Text706), ADR(gc_DbmTranslation_en_Text707), ADR(gc_DbmTranslation_en_Text708), ADR(gc_DbmTranslation_en_Text709), ADR(gc_DbmTranslation_en_Text710), ADR(gc_DbmTranslation_en_Text711), ADR(gc_DbmTranslation_en_Text712), ADR(gc_DbmTranslation_en_Text713), ADR(gc_DbmTranslation_en_Text714), ADR(gc_DbmTranslation_en_Text715), ADR(gc_DbmTranslation_en_Text716), ADR(gc_DbmTranslation_en_Text717), ADR(gc_DbmTranslation_en_Text718), ADR(gc_DbmTranslation_en_Text719), ADR(gc_DbmTranslation_en_Text720), ADR(gc_DbmTranslation_en_Text721), ADR(gc_DbmTranslation_en_Text722), ADR(gc_DbmTranslation_en_Text723), ADR(gc_DbmTranslation_en_Text724), ADR(gc_DbmTranslation_en_Text725), ADR(gc_DbmTranslation_en_Text726), ADR(gc_DbmTranslation_en_Text727), ADR(gc_DbmTranslation_en_Text728), ADR(gc_DbmTranslation_en_Text729), ADR(gc_DbmTranslation_en_Text730), ADR(gc_DbmTranslation_en_Text731), ADR(gc_DbmTranslation_en_Text732), ADR(gc_DbmTranslation_en_Text733), ADR(gc_DbmTranslation_en_Text734), ADR(gc_DbmTranslation_en_Text735), ADR(gc_DbmTranslation_en_Text736), ADR(gc_DbmTranslation_en_Text737), ADR(gc_DbmTranslation_en_Text738), ADR(gc_DbmTranslation_en_Text739), ADR(gc_DbmTranslation_en_Text740), ADR(gc_DbmTranslation_en_Text741), ADR(gc_DbmTranslation_en_Text742), ADR(gc_DbmTranslation_en_Text743), ADR(gc_DbmTranslation_en_Text744), ADR(gc_DbmTranslation_en_Text745), ADR(gc_DbmTranslation_en_Text746), ADR(gc_DbmTranslation_en_Text747), ADR(gc_DbmTranslation_en_Text748), ADR(gc_DbmTranslation_en_Text749), ADR(gc_DbmTranslation_en_Text750), ADR(gc_DbmTranslation_en_Text751), ADR(gc_DbmTranslation_en_Text752), ADR(gc_DbmTranslation_en_Text753), ADR(gc_DbmTranslation_en_Text754), ADR(gc_DbmTranslation_en_Text755), ADR(gc_DbmTranslation_en_Text756), ADR(gc_DbmTranslation_en_Text757), ADR(gc_DbmTranslation_en_Text758), ADR(gc_DbmTranslation_en_Text759), ADR(gc_DbmTranslation_en_Text760), ADR(gc_DbmTranslation_en_Text761), ADR(gc_DbmTranslation_en_Text762), ADR(gc_DbmTranslation_en_Text763), ADR(gc_DbmTranslation_en_Text764), ADR(gc_DbmTranslation_en_Text765), ADR(gc_DbmTranslation_en_Text766), ADR(gc_DbmTranslation_en_Text767), ADR(gc_DbmTranslation_en_Text768), ADR(gc_DbmTranslation_en_Text769), ADR(gc_DbmTranslation_en_Text770), ADR(gc_DbmTranslation_en_Text771), ADR(gc_DbmTranslation_en_Text772), ADR(gc_DbmTranslation_en_Text773), ADR(gc_DbmTranslation_en_Text774), ADR(gc_DbmTranslation_en_Text775), ADR(gc_DbmTranslation_en_Text776), ADR(gc_DbmTranslation_en_Text777), ADR(gc_DbmTranslation_en_Text778), ADR(gc_DbmTranslation_en_Text779), ADR(gc_DbmTranslation_en_Text780), ADR(gc_DbmTranslation_en_Text781), ADR(gc_DbmTranslation_en_Text782), ADR(gc_DbmTranslation_en_Text783), ADR(gc_DbmTranslation_en_Text784), ADR(gc_DbmTranslation_en_Text785), ADR(gc_DbmTranslation_en_Text786), ADR(gc_DbmTranslation_en_Text787), ADR(gc_DbmTranslation_en_Text788), ADR(gc_DbmTranslation_en_Text789), ADR(gc_DbmTranslation_en_Text790), ADR(gc_DbmTranslation_en_Text791), ADR(gc_DbmTranslation_en_Text792), ADR(gc_DbmTranslation_en_Text793), ADR(gc_DbmTranslation_en_Text794), ADR(gc_DbmTranslation_en_Text795), ADR(gc_DbmTranslation_en_Text796), ADR(gc_DbmTranslation_en_Text797), ADR(gc_DbmTranslation_en_Text798), ADR(gc_DbmTranslation_en_Text799), ADR(gc_DbmTranslation_en_Text800), ADR(gc_DbmTranslation_en_Text801), ADR(gc_DbmTranslation_en_Text802), ADR(gc_DbmTranslation_en_Text803), ADR(gc_DbmTranslation_en_Text804), ADR(gc_DbmTranslation_en_Text805), ADR(gc_DbmTranslation_en_Text806), ADR(gc_DbmTranslation_en_Text807), ADR(gc_DbmTranslation_en_Text808), ADR(gc_DbmTranslation_en_Text809), ADR(gc_DbmTranslation_en_Text810), ADR(gc_DbmTranslation_en_Text811), ADR(gc_DbmTranslation_en_Text812), ADR(gc_DbmTranslation_en_Text813), ADR(gc_DbmTranslation_en_Text814), ADR(gc_DbmTranslation_en_Text815), ADR(gc_DbmTranslation_en_Text816), ADR(gc_DbmTranslation_en_Text817), ADR(gc_DbmTranslation_en_Text818), ADR(gc_DbmTranslation_en_Text819), ADR(gc_DbmTranslation_en_Text820), ADR(gc_DbmTranslation_en_Text821), ADR(gc_DbmTranslation_en_Text822), ADR(gc_DbmTranslation_en_Text823), ADR(gc_DbmTranslation_en_Text824), ADR(gc_DbmTranslation_en_Text825), ADR(gc_DbmTranslation_en_Text826), ADR(gc_DbmTranslation_en_Text827), ADR(gc_DbmTranslation_en_Text828), ADR(gc_DbmTranslation_en_Text829), ADR(gc_DbmTranslation_en_Text830), ADR(gc_DbmTranslation_en_Text831), ADR(gc_DbmTranslation_en_Text832), ADR(gc_DbmTranslation_en_Text833), ADR(gc_DbmTranslation_en_Text834), ADR(gc_DbmTranslation_en_Text835), ADR(gc_DbmTranslation_en_Text836), ADR(gc_DbmTranslation_en_Text837), ADR(gc_DbmTranslation_en_Text838), ADR(gc_DbmTranslation_en_Text839), ADR(gc_DbmTranslation_en_Text840), ADR(gc_DbmTranslation_en_Text841), ADR(gc_DbmTranslation_en_Text842), ADR(gc_DbmTranslation_en_Text843), ADR(gc_DbmTranslation_en_Text844), ADR(gc_DbmTranslation_en_Text845), ADR(gc_DbmTranslation_en_Text846), ADR(gc_DbmTranslation_en_Text847), ADR(gc_DbmTranslation_en_Text848), ADR(gc_DbmTranslation_en_Text849), ADR(gc_DbmTranslation_en_Text850), ADR(gc_DbmTranslation_en_Text851), ADR(gc_DbmTranslation_en_Text852), ADR(gc_DbmTranslation_en_Text853), ADR(gc_DbmTranslation_en_Text854), ADR(gc_DbmTranslation_en_Text855), ADR(gc_DbmTranslation_en_Text856), ADR(gc_DbmTranslation_en_Text857), ADR(gc_DbmTranslation_en_Text858), ADR(gc_DbmTranslation_en_Text859), ADR(gc_DbmTranslation_en_Text860), ADR(gc_DbmTranslation_en_Text861), ADR(gc_DbmTranslation_en_Text862), ADR(gc_DbmTranslation_en_Text863), ADR(gc_DbmTranslation_en_Text864), ADR(gc_DbmTranslation_en_Text865), ADR(gc_DbmTranslation_en_Text866), ADR(gc_DbmTranslation_en_Text867), ADR(gc_DbmTranslation_en_Text868), ADR(gc_DbmTranslation_en_Text869), ADR(gc_DbmTranslation_en_Text870), ADR(gc_DbmTranslation_en_Text871), ADR(gc_DbmTranslation_en_Text872), ADR(gc_DbmTranslation_en_Text873), ADR(gc_DbmTranslation_en_Text874), ADR(gc_DbmTranslation_en_Text875), ADR(gc_DbmTranslation_en_Text876), ADR(gc_DbmTranslation_en_Text877), ADR(gc_DbmTranslation_en_Text878), ADR(gc_DbmTranslation_en_Text879), ADR(gc_DbmTranslation_en_Text880), ADR(gc_DbmTranslation_en_Text881), ADR(gc_DbmTranslation_en_Text882), ADR(gc_DbmTranslation_en_Text883), ADR(gc_DbmTranslation_en_Text884), ADR(gc_DbmTranslation_en_Text885), ADR(gc_DbmTranslation_en_Text886), ADR(gc_DbmTranslation_en_Text887), ADR(gc_DbmTranslation_en_Text888), ADR(gc_DbmTranslation_en_Text889), ADR(gc_DbmTranslation_en_Text890), ADR(gc_DbmTranslation_en_Text891), ADR(gc_DbmTranslation_en_Text892), ADR(gc_DbmTranslation_en_Text893), ADR(gc_DbmTranslation_en_Text894), ADR(gc_DbmTranslation_en_Text895), ADR(gc_DbmTranslation_en_Text896), ADR(gc_DbmTranslation_en_Text897), ADR(gc_DbmTranslation_en_Text898), ADR(gc_DbmTranslation_en_Text899), ADR(gc_DbmTranslation_en_Text900), ADR(gc_DbmTranslation_en_Text901), ADR(gc_DbmTranslation_en_Text902), ADR(gc_DbmTranslation_en_Text903), ADR(gc_DbmTranslation_en_Text904), ADR(gc_DbmTranslation_en_Text905), ADR(gc_DbmTranslation_en_Text906), ADR(gc_DbmTranslation_en_Text907), ADR(gc_DbmTranslation_en_Text908), ADR(gc_DbmTranslation_en_Text909), ADR(gc_DbmTranslation_en_Text910), ADR(gc_DbmTranslation_en_Text911), ADR(gc_DbmTranslation_en_Text912), ADR(gc_DbmTranslation_en_Text913), ADR(gc_DbmTranslation_en_Text914), ADR(gc_DbmTranslation_en_Text915), ADR(gc_DbmTranslation_en_Text916), ADR(gc_DbmTranslation_en_Text917), ADR(gc_DbmTranslation_en_Text918), ADR(gc_DbmTranslation_en_Text919), ADR(gc_DbmTranslation_en_Text920), ADR(gc_DbmTranslation_en_Text921), ADR(gc_DbmTranslation_en_Text922), ADR(gc_DbmTranslation_en_Text923), ADR(gc_DbmTranslation_en_Text924), ADR(gc_DbmTranslation_en_Text925), ADR(gc_DbmTranslation_en_Text926), ADR(gc_DbmTranslation_en_Text927), ADR(gc_DbmTranslation_en_Text928), ADR(gc_DbmTranslation_en_Text929), ADR(gc_DbmTranslation_en_Text930), ADR(gc_DbmTranslation_en_Text931), ADR(gc_DbmTranslation_en_Text932), ADR(gc_DbmTranslation_en_Text933), ADR(gc_DbmTranslation_en_Text934), ADR(gc_DbmTranslation_en_Text935), ADR(gc_DbmTranslation_en_Text936), ADR(gc_DbmTranslation_en_Text937), ADR(gc_DbmTranslation_en_Text938), ADR(gc_DbmTranslation_en_Text939), ADR(gc_DbmTranslation_en_Text940), ADR(gc_DbmTranslation_en_Text941), ADR(gc_DbmTranslation_en_Text942), ADR(gc_DbmTranslation_en_Text943), ADR(gc_DbmTranslation_en_Text944), ADR(gc_DbmTranslation_en_Text945), ADR(gc_DbmTranslation_en_Text946), ADR(gc_DbmTranslation_en_Text947), ADR(gc_DbmTranslation_en_Text948), ADR(gc_DbmTranslation_en_Text949), ADR(gc_DbmTranslation_en_Text950), ADR(gc_DbmTranslation_en_Text951), ADR(gc_DbmTranslation_en_Text952), ADR(gc_DbmTranslation_en_Text953), ADR(gc_DbmTranslation_en_Text954), ADR(gc_DbmTranslation_en_Text955), ADR(gc_DbmTranslation_en_Text956), ADR(gc_DbmTranslation_en_Text957), ADR(gc_DbmTranslation_en_Text958), ADR(gc_DbmTranslation_en_Text959), ADR(gc_DbmTranslation_en_Text960), ADR(gc_DbmTranslation_en_Text961), ADR(gc_DbmTranslation_en_Text962), ADR(gc_DbmTranslation_en_Text963), ADR(gc_DbmTranslation_en_Text964), ADR(gc_DbmTranslation_en_Text965), ADR(gc_DbmTranslation_en_Text966), ADR(gc_DbmTranslation_en_Text967), ADR(gc_DbmTranslation_en_Text968), ADR(gc_DbmTranslation_en_Text969), ADR(gc_DbmTranslation_en_Text970), ADR(gc_DbmTranslation_en_Text971), ADR(gc_DbmTranslation_en_Text972), ADR(gc_DbmTranslation_en_Text973), ADR(gc_DbmTranslation_en_Text974), ADR(gc_DbmTranslation_en_Text975), ADR(gc_DbmTranslation_en_Text976), ADR(gc_DbmTranslation_en_Text977), ADR(gc_DbmTranslation_en_Text978), ADR(gc_DbmTranslation_en_Text979), ADR(gc_DbmTranslation_en_Text980), ADR(gc_DbmTranslation_en_Text981), ADR(gc_DbmTranslation_en_Text982), ADR(gc_DbmTranslation_en_Text983), ADR(gc_DbmTranslation_en_Text984), ADR(gc_DbmTranslation_en_Text985), ADR(gc_DbmTranslation_en_Text986), ADR(gc_DbmTranslation_en_Text987), ADR(gc_DbmTranslation_en_Text988), ADR(gc_DbmTranslation_en_Text989), ADR(gc_DbmTranslation_en_Text990), ADR(gc_DbmTranslation_en_Text991), ADR(gc_DbmTranslation_en_Text992), ADR(gc_DbmTranslation_en_Text993), ADR(gc_DbmTranslation_en_Text994), ADR(gc_DbmTranslation_en_Text995), ADR(gc_DbmTranslation_en_Text996), ADR(gc_DbmTranslation_en_Text997), ADR(gc_DbmTranslation_en_Text998), ADR(gc_DbmTranslation_en_Text999), ADR(gc_DbmTranslation_en_Text1000), ADR(gc_DbmTranslation_en_Text1001), ADR(gc_DbmTranslation_en_Text1002), ADR(gc_DbmTranslation_en_Text1003), ADR(gc_DbmTranslation_en_Text1004), ADR(gc_DbmTranslation_en_Text1005), ADR(gc_DbmTranslation_en_Text1006), ADR(gc_DbmTranslation_en_Text1007), ADR(gc_DbmTranslation_en_Text1008), ADR(gc_DbmTranslation_en_Text1009), ADR(gc_DbmTranslation_en_Text1010), ADR(gc_DbmTranslation_en_Text1011), ADR(gc_DbmTranslation_en_Text1012), ADR(gc_DbmTranslation_en_Text1013), ADR(gc_DbmTranslation_en_Text1014), ADR(gc_DbmTranslation_en_Text1015), ADR(gc_DbmTranslation_en_Text1016), ADR(gc_DbmTranslation_en_Text1017), ADR(gc_DbmTranslation_en_Text1018), ADR(gc_DbmTranslation_en_Text1019), ADR(gc_DbmTranslation_en_Text1020), ADR(gc_DbmTranslation_en_Text1021), ADR(gc_DbmTranslation_en_Text1022), ADR(gc_DbmTranslation_en_Text1023), ADR(gc_DbmTranslation_en_Text1024), ADR(gc_DbmTranslation_en_Text1025), ADR(gc_DbmTranslation_en_Text1026), ADR(gc_DbmTranslation_en_Text1027), ADR(gc_DbmTranslation_en_Text1028), ADR(gc_DbmTranslation_en_Text1029), ADR(gc_DbmTranslation_en_Text1030), ADR(gc_DbmTranslation_en_Text1031), ADR(gc_DbmTranslation_en_Text1032), ADR(gc_DbmTranslation_en_Text1033), ADR(gc_DbmTranslation_en_Text1034), ADR(gc_DbmTranslation_en_Text1035), ADR(gc_DbmTranslation_en_Text1036), ADR(gc_DbmTranslation_en_Text1037), ADR(gc_DbmTranslation_en_Text1038), ADR(gc_DbmTranslation_en_Text1039), ADR(gc_DbmTranslation_en_Text1040), ADR(gc_DbmTranslation_en_Text1041), ADR(gc_DbmTranslation_en_Text1042), ADR(gc_DbmTranslation_en_Text1043), ADR(gc_DbmTranslation_en_Text1044), ADR(gc_DbmTranslation_en_Text1045), ADR(gc_DbmTranslation_en_Text1046), ADR(gc_DbmTranslation_en_Text1047), ADR(gc_DbmTranslation_en_Text1048), ADR(gc_DbmTranslation_en_Text1049), ADR(gc_DbmTranslation_en_Text1050), ADR(gc_DbmTranslation_en_Text1051), ADR(gc_DbmTranslation_en_Text1052), ADR(gc_DbmTranslation_en_Text1053), ADR(gc_DbmTranslation_en_Text1054), ADR(gc_DbmTranslation_en_Text1055), ADR(gc_DbmTranslation_en_Text1056), ADR(gc_DbmTranslation_en_Text1057), ADR(gc_DbmTranslation_en_Text1058), ADR(gc_DbmTranslation_en_Text1059), ADR(gc_DbmTranslation_en_Text1060), ADR(gc_DbmTranslation_en_Text1061), ADR(gc_DbmTranslation_en_Text1062), ADR(gc_DbmTranslation_en_Text1063), ADR(gc_DbmTranslation_en_Text1064), ADR(gc_DbmTranslation_en_Text1065), ADR(gc_DbmTranslation_en_Text1066), ADR(gc_DbmTranslation_en_Text1067), ADR(gc_DbmTranslation_en_Text1068), ADR(gc_DbmTranslation_en_Text1069), ADR(gc_DbmTranslation_en_Text1070), ADR(gc_DbmTranslation_en_Text1071), ADR(gc_DbmTranslation_en_Text1072), ADR(gc_DbmTranslation_en_Text1073), ADR(gc_DbmTranslation_en_Text1074), ADR(gc_DbmTranslation_en_Text1075), ADR(gc_DbmTranslation_en_Text1076), ADR(gc_DbmTranslation_en_Text1077), ADR(gc_DbmTranslation_en_Text1078), ADR(gc_DbmTranslation_en_Text1079), ADR(gc_DbmTranslation_en_Text1080), ADR(gc_DbmTranslation_en_Text1081), ADR(gc_DbmTranslation_en_Text1082), ADR(gc_DbmTranslation_en_Text1083), ADR(gc_DbmTranslation_en_Text1084), ADR(gc_DbmTranslation_en_Text1085), ADR(gc_DbmTranslation_en_Text1086), ADR(gc_DbmTranslation_en_Text1087), ADR(gc_DbmTranslation_en_Text1088), ADR(gc_DbmTranslation_en_Text1089), ADR(gc_DbmTranslation_en_Text1090), ADR(gc_DbmTranslation_en_Text1091), ADR(gc_DbmTranslation_en_Text1092), ADR(gc_DbmTranslation_en_Text1093), ADR(gc_DbmTranslation_en_Text1094), ADR(gc_DbmTranslation_en_Text1095), ADR(gc_DbmTranslation_en_Text1096), ADR(gc_DbmTranslation_en_Text1097), ADR(gc_DbmTranslation_en_Text1098), ADR(gc_DbmTranslation_en_Text1099), ADR(gc_DbmTranslation_en_Text1100), ADR(gc_DbmTranslation_en_Text1101), ADR(gc_DbmTranslation_en_Text1102), ADR(gc_DbmTranslation_en_Text1103), ADR(gc_DbmTranslation_en_Text1104), ADR(gc_DbmTranslation_en_Text1105), ADR(gc_DbmTranslation_en_Text1106), ADR(gc_DbmTranslation_en_Text1107), ADR(gc_DbmTranslation_en_Text1108), ADR(gc_DbmTranslation_en_Text1109), ADR(gc_DbmTranslation_en_Text1110), ADR(gc_DbmTranslation_en_Text1111), ADR(gc_DbmTranslation_en_Text1112), ADR(gc_DbmTranslation_en_Text1113), ADR(gc_DbmTranslation_en_Text1114), ADR(gc_DbmTranslation_en_Text1115), ADR(gc_DbmTranslation_en_Text1116), ADR(gc_DbmTranslation_en_Text1117), ADR(gc_DbmTranslation_en_Text1118), ADR(gc_DbmTranslation_en_Text1119), ADR(gc_DbmTranslation_en_Text1120), ADR(gc_DbmTranslation_en_Text1121), ADR(gc_DbmTranslation_en_Text1122), ADR(gc_DbmTranslation_en_Text1123), ADR(gc_DbmTranslation_en_Text1124), ADR(gc_DbmTranslation_en_Text1125), ADR(gc_DbmTranslation_en_Text1126), ADR(gc_DbmTranslation_en_Text1127), ADR(gc_DbmTranslation_en_Text1128), ADR(gc_DbmTranslation_en_Text1129), ADR(gc_DbmTranslation_en_Text1130), ADR(gc_DbmTranslation_en_Text1131), ADR(gc_DbmTranslation_en_Text1132), ADR(gc_DbmTranslation_en_Text1133), ADR(gc_DbmTranslation_en_Text1134), ADR(gc_DbmTranslation_en_Text1135), ADR(gc_DbmTranslation_en_Text1136), ADR(gc_DbmTranslation_en_Text1137), ADR(gc_DbmTranslation_en_Text1138), ADR(gc_DbmTranslation_en_Text1139), ADR(gc_DbmTranslation_en_Text1140), ADR(gc_DbmTranslation_en_Text1141), ADR(gc_DbmTranslation_en_Text1142), ADR(gc_DbmTranslation_en_Text1143), ADR(gc_DbmTranslation_en_Text1144), ADR(gc_DbmTranslation_en_Text1145), ADR(gc_DbmTranslation_en_Text1146), ADR(gc_DbmTranslation_en_Text1147), ADR(gc_DbmTranslation_en_Text1148), ADR(gc_DbmTranslation_en_Text1149), ADR(gc_DbmTranslation_en_Text1150), ADR(gc_DbmTranslation_en_Text1151), ADR(gc_DbmTranslation_en_Text1152), ADR(gc_DbmTranslation_en_Text1153), ADR(gc_DbmTranslation_en_Text1154), ADR(gc_DbmTranslation_en_Text1155), ADR(gc_DbmTranslation_en_Text1156), ADR(gc_DbmTranslation_en_Text1157), ADR(gc_DbmTranslation_en_Text1158), ADR(gc_DbmTranslation_en_Text1159), ADR(gc_DbmTranslation_en_Text1160), ADR(gc_DbmTranslation_en_Text1161), ADR(gc_DbmTranslation_en_Text1162), ADR(gc_DbmTranslation_en_Text1163), ADR(gc_DbmTranslation_en_Text1164), ADR(gc_DbmTranslation_en_Text1165), ADR(gc_DbmTranslation_en_Text1166), ADR(gc_DbmTranslation_en_Text1167), ADR(gc_DbmTranslation_en_Text1168), ADR(gc_DbmTranslation_en_Text1169), ADR(gc_DbmTranslation_en_Text1170), ADR(gc_DbmTranslation_en_Text1171), ADR(gc_DbmTranslation_en_Text1172), ADR(gc_DbmTranslation_en_Text1173), ADR(gc_DbmTranslation_en_Text1174), ADR(gc_DbmTranslation_en_Text1175), ADR(gc_DbmTranslation_en_Text1176), ADR(gc_DbmTranslation_en_Text1177), ADR(gc_DbmTranslation_en_Text1178), ADR(gc_DbmTranslation_en_Text1179), ADR(gc_DbmTranslation_en_Text1180), ADR(gc_DbmTranslation_en_Text1181), ADR(gc_DbmTranslation_en_Text1182), ADR(gc_DbmTranslation_en_Text1183), ADR(gc_DbmTranslation_en_Text1184), ADR(gc_DbmTranslation_en_Text1185), ADR(gc_DbmTranslation_en_Text1186), ADR(gc_DbmTranslation_en_Text1187), ADR(gc_DbmTranslation_en_Text1188), ADR(gc_DbmTranslation_en_Text1189), ADR(gc_DbmTranslation_en_Text1190), ADR(gc_DbmTranslation_en_Text1191), ADR(gc_DbmTranslation_en_Text1192), ADR(gc_DbmTranslation_en_Text1193), ADR(gc_DbmTranslation_en_Text1194), ADR(gc_DbmTranslation_en_Text1195), ADR(gc_DbmTranslation_en_Text1196), ADR(gc_DbmTranslation_en_Text1197), ADR(gc_DbmTranslation_en_Text1198), ADR(gc_DbmTranslation_en_Text1199), ADR(gc_DbmTranslation_en_Text1200), ADR(gc_DbmTranslation_en_Text1201), ADR(gc_DbmTranslation_en_Text1202), ADR(gc_DbmTranslation_en_Text1203), ADR(gc_DbmTranslation_en_Text1204), ADR(gc_DbmTranslation_en_Text1205), ADR(gc_DbmTranslation_en_Text1206), ADR(gc_DbmTranslation_en_Text1207), ADR(gc_DbmTranslation_en_Text1208), ADR(gc_DbmTranslation_en_Text1209), ADR(gc_DbmTranslation_en_Text1210), ADR(gc_DbmTranslation_en_Text1211), ADR(gc_DbmTranslation_en_Text1212), ADR(gc_DbmTranslation_en_Text1213), ADR(gc_DbmTranslation_en_Text1214), ADR(gc_DbmTranslation_en_Text1215), ADR(gc_DbmTranslation_en_Text1216), ADR(gc_DbmTranslation_en_Text1217), ADR(gc_DbmTranslation_en_Text1218), ADR(gc_DbmTranslation_en_Text1219), ADR(gc_DbmTranslation_en_Text1220), ADR(gc_DbmTranslation_en_Text1221), ADR(gc_DbmTranslation_en_Text1222), ADR(gc_DbmTranslation_en_Text1223), ADR(gc_DbmTranslation_en_Text1224), ADR(gc_DbmTranslation_en_Text1225), ADR(gc_DbmTranslation_en_Text1226), ADR(gc_DbmTranslation_en_Text1227), ADR(gc_DbmTranslation_en_Text1228), ADR(gc_DbmTranslation_en_Text1229), ADR(gc_DbmTranslation_en_Text1230), ADR(gc_DbmTranslation_en_Text1231), ADR(gc_DbmTranslation_en_Text1232), ADR(gc_DbmTranslation_en_Text1233), ADR(gc_DbmTranslation_en_Text1234), ADR(gc_DbmTranslation_en_Text1235), ADR(gc_DbmTranslation_en_Text1236), ADR(gc_DbmTranslation_en_Text1237), ADR(gc_DbmTranslation_en_Text1238), ADR(gc_DbmTranslation_en_Text1239), ADR(gc_DbmTranslation_en_Text1240), ADR(gc_DbmTranslation_en_Text1241), ADR(gc_DbmTranslation_en_Text1242), ADR(gc_DbmTranslation_en_Text1243), ADR(gc_DbmTranslation_en_Text1244), ADR(gc_DbmTranslation_en_Text1245), ADR(gc_DbmTranslation_en_Text1246), ADR(gc_DbmTranslation_en_Text1247), ADR(gc_DbmTranslation_en_Text1248), ADR(gc_DbmTranslation_en_Text1249), ADR(gc_DbmTranslation_en_Text1250), ADR(gc_DbmTranslation_en_Text1251), ADR(gc_DbmTranslation_en_Text1252), ADR(gc_DbmTranslation_en_Text1253), ADR(gc_DbmTranslation_en_Text1254), ADR(gc_DbmTranslation_en_Text1255), ADR(gc_DbmTranslation_en_Text1256), ADR(gc_DbmTranslation_en_Text1257), ADR(gc_DbmTranslation_en_Text1258), ADR(gc_DbmTranslation_en_Text1259), ADR(gc_DbmTranslation_en_Text1260), ADR(gc_DbmTranslation_en_Text1261), ADR(gc_DbmTranslation_en_Text1262), ADR(gc_DbmTranslation_en_Text1263), ADR(gc_DbmTranslation_en_Text1264), ADR(gc_DbmTranslation_en_Text1265), ADR(gc_DbmTranslation_en_Text1266), ADR(gc_DbmTranslation_en_Text1267), ADR(gc_DbmTranslation_en_Text1268), ADR(gc_DbmTranslation_en_Text1269), ADR(gc_DbmTranslation_en_Text1270), ADR(gc_DbmTranslation_en_Text1271), ADR(gc_DbmTranslation_en_Text1272), ADR(gc_DbmTranslation_en_Text1273), ADR(gc_DbmTranslation_en_Text1274), ADR(gc_DbmTranslation_en_Text1275), ADR(gc_DbmTranslation_en_Text1276), ADR(gc_DbmTranslation_en_Text1277), ADR(gc_DbmTranslation_en_Text1278), ADR(gc_DbmTranslation_en_Text1279), ADR(gc_DbmTranslation_en_Text1280), ADR(gc_DbmTranslation_en_Text1281), ADR(gc_DbmTranslation_en_Text1282), ADR(gc_DbmTranslation_en_Text1283), ADR(gc_DbmTranslation_en_Text1284), ADR(gc_DbmTranslation_en_Text1285), ADR(gc_DbmTranslation_en_Text1286), ADR(gc_DbmTranslation_en_Text1287), ADR(gc_DbmTranslation_en_Text1288), ADR(gc_DbmTranslation_en_Text1289), ADR(gc_DbmTranslation_en_Text1290), ADR(gc_DbmTranslation_en_Text1291), ADR(gc_DbmTranslation_en_Text1292), ADR(gc_DbmTranslation_en_Text1293), ADR(gc_DbmTranslation_en_Text1294), ADR(gc_DbmTranslation_en_Text1295), ADR(gc_DbmTranslation_en_Text1296), ADR(gc_DbmTranslation_en_Text1297), ADR(gc_DbmTranslation_en_Text1298), ADR(gc_DbmTranslation_en_Text1299), ADR(gc_DbmTranslation_en_Text1300), ADR(gc_DbmTranslation_en_Text1301), ADR(gc_DbmTranslation_en_Text1302), ADR(gc_DbmTranslation_en_Text1303), ADR(gc_DbmTranslation_en_Text1304), ADR(gc_DbmTranslation_en_Text1305), ADR(gc_DbmTranslation_en_Text1306), ADR(gc_DbmTranslation_en_Text1307), ADR(gc_DbmTranslation_en_Text1308), ADR(gc_DbmTranslation_en_Text1309), ADR(gc_DbmTranslation_en_Text1310), ADR(gc_DbmTranslation_en_Text1311), ADR(gc_DbmTranslation_en_Text1312), ADR(gc_DbmTranslation_en_Text1313), ADR(gc_DbmTranslation_en_Text1314), ADR(gc_DbmTranslation_en_Text1315), ADR(gc_DbmTranslation_en_Text1316), ADR(gc_DbmTranslation_en_Text1317), ADR(gc_DbmTranslation_en_Text1318), ADR(gc_DbmTranslation_en_Text1319), ADR(gc_DbmTranslation_en_Text1320), ADR(gc_DbmTranslation_en_Text1321), ADR(gc_DbmTranslation_en_Text1322), ADR(gc_DbmTranslation_en_Text1323), ADR(gc_DbmTranslation_en_Text1324), ADR(gc_DbmTranslation_en_Text1325), ADR(gc_DbmTranslation_en_Text1326), ADR(gc_DbmTranslation_en_Text1327), ADR(gc_DbmTranslation_en_Text1328), ADR(gc_DbmTranslation_en_Text1329), ADR(gc_DbmTranslation_en_Text1330), ADR(gc_DbmTranslation_en_Text1331), ADR(gc_DbmTranslation_en_Text1332), ADR(gc_DbmTranslation_en_Text1333), ADR(gc_DbmTranslation_en_Text1334), ADR(gc_DbmTranslation_en_Text1335), ADR(gc_DbmTranslation_en_Text1336), ADR(gc_DbmTranslation_en_Text1337), ADR(gc_DbmTranslation_en_Text1338), ADR(gc_DbmTranslation_en_Text1339), ADR(gc_DbmTranslation_en_Text1340), ADR(gc_DbmTranslation_en_Text1341), ADR(gc_DbmTranslation_en_Text1342), ADR(gc_DbmTranslation_en_Text1343), ADR(gc_DbmTranslation_en_Text1344), ADR(gc_DbmTranslation_en_Text1345), ADR(gc_DbmTranslation_en_Text1346), ADR(gc_DbmTranslation_en_Text1347), ADR(gc_DbmTranslation_en_Text1348), ADR(gc_DbmTranslation_en_Text1349), ADR(gc_DbmTranslation_en_Text1350), ADR(gc_DbmTranslation_en_Text1351), ADR(gc_DbmTranslation_en_Text1352), ADR(gc_DbmTranslation_en_Text1353), ADR(gc_DbmTranslation_en_Text1354), ADR(gc_DbmTranslation_en_Text1355), ADR(gc_DbmTranslation_en_Text1356), ADR(gc_DbmTranslation_en_Text1357), ADR(gc_DbmTranslation_en_Text1358), ADR(gc_DbmTranslation_en_Text1359), ADR(gc_DbmTranslation_en_Text1360), ADR(gc_DbmTranslation_en_Text1361), ADR(gc_DbmTranslation_en_Text1362), ADR(gc_DbmTranslation_en_Text1363), ADR(gc_DbmTranslation_en_Text1364), ADR(gc_DbmTranslation_en_Text1365), ADR(gc_DbmTranslation_en_Text1366), ADR(gc_DbmTranslation_en_Text1367), ADR(gc_DbmTranslation_en_Text1368), ADR(gc_DbmTranslation_en_Text1369), ADR(gc_DbmTranslation_en_Text1370), ADR(gc_DbmTranslation_en_Text1371), ADR(gc_DbmTranslation_en_Text1372), ADR(gc_DbmTranslation_en_Text1373), ADR(gc_DbmTranslation_en_Text1374), ADR(gc_DbmTranslation_en_Text1375), ADR(gc_DbmTranslation_en_Text1376), ADR(gc_DbmTranslation_en_Text1377), ADR(gc_DbmTranslation_en_Text1378), ADR(gc_DbmTranslation_en_Text1379), ADR(gc_DbmTranslation_en_Text1380), ADR(gc_DbmTranslation_en_Text1381), ADR(gc_DbmTranslation_en_Text1382), ADR(gc_DbmTranslation_en_Text1383), ADR(gc_DbmTranslation_en_Text1384), ADR(gc_DbmTranslation_en_Text1385), ADR(gc_DbmTranslation_en_Text1386), ADR(gc_DbmTranslation_en_Text1387), ADR(gc_DbmTranslation_en_Text1388), ADR(gc_DbmTranslation_en_Text1389), ADR(gc_DbmTranslation_en_Text1390), ADR(gc_DbmTranslation_en_Text1391), ADR(gc_DbmTranslation_en_Text1392), ADR(gc_DbmTranslation_en_Text1393), ADR(gc_DbmTranslation_en_Text1394), ADR(gc_DbmTranslation_en_Text1395), ADR(gc_DbmTranslation_en_Text1396), ADR(gc_DbmTranslation_en_Text1397), ADR(gc_DbmTranslation_en_Text1398), ADR(gc_DbmTranslation_en_Text1399), ADR(gc_DbmTranslation_en_Text1400), ADR(gc_DbmTranslation_en_Text1401), ADR(gc_DbmTranslation_en_Text1402), ADR(gc_DbmTranslation_en_Text1403), ADR(gc_DbmTranslation_en_Text1404), ADR(gc_DbmTranslation_en_Text1405), ADR(gc_DbmTranslation_en_Text1406), ADR(gc_DbmTranslation_en_Text1407), ADR(gc_DbmTranslation_en_Text1408), ADR(gc_DbmTranslation_en_Text1409), ADR(gc_DbmTranslation_en_Text1410), ADR(gc_DbmTranslation_en_Text1411), ADR(gc_DbmTranslation_en_Text1412), ADR(gc_DbmTranslation_en_Text1413), ADR(gc_DbmTranslation_en_Text1414), ADR(gc_DbmTranslation_en_Text1415), ADR(gc_DbmTranslation_en_Text1416), ADR(gc_DbmTranslation_en_Text1417), ADR(gc_DbmTranslation_en_Text1418), ADR(gc_DbmTranslation_en_Text1419), ADR(gc_DbmTranslation_en_Text1420), ADR(gc_DbmTranslation_en_Text1421), ADR(gc_DbmTranslation_en_Text1422), ADR(gc_DbmTranslation_en_Text1423), ADR(gc_DbmTranslation_en_Text1424), ADR(gc_DbmTranslation_en_Text1425), ADR(gc_DbmTranslation_en_Text1426), ADR(gc_DbmTranslation_en_Text1427), ADR(gc_DbmTranslation_en_Text1428), ADR(gc_DbmTranslation_en_Text1429), ADR(gc_DbmTranslation_en_Text1430), ADR(gc_DbmTranslation_en_Text1431), ADR(gc_DbmTranslation_en_Text1432), ADR(gc_DbmTranslation_en_Text1433), ADR(gc_DbmTranslation_en_Text1434), ADR(gc_DbmTranslation_en_Text1435), ADR(gc_DbmTranslation_en_Text1436), ADR(gc_DbmTranslation_en_Text1437), ADR(gc_DbmTranslation_en_Text1438), ADR(gc_DbmTranslation_en_Text1439), ADR(gc_DbmTranslation_en_Text1440), ADR(gc_DbmTranslation_en_Text1441), ADR(gc_DbmTranslation_en_Text1442), ADR(gc_DbmTranslation_en_Text1443), ADR(gc_DbmTranslation_en_Text1444), ADR(gc_DbmTranslation_en_Text1445), ADR(gc_DbmTranslation_en_Text1446), ADR(gc_DbmTranslation_en_Text1447), ADR(gc_DbmTranslation_en_Text1448), ADR(gc_DbmTranslation_en_Text1449), ADR(gc_DbmTranslation_en_Text1450), ADR(gc_DbmTranslation_en_Text1451), ADR(gc_DbmTranslation_en_Text1452), ADR(gc_DbmTranslation_en_Text1453), ADR(gc_DbmTranslation_en_Text1454), ADR(gc_DbmTranslation_en_Text1455), ADR(gc_DbmTranslation_en_Text1456), ADR(gc_DbmTranslation_en_Text1457), ADR(gc_DbmTranslation_en_Text1458), ADR(gc_DbmTranslation_en_Text1459), ADR(gc_DbmTranslation_en_Text1460), ADR(gc_DbmTranslation_en_Text1461), ADR(gc_DbmTranslation_en_Text1462), ADR(gc_DbmTranslation_en_Text1463), ADR(gc_DbmTranslation_en_Text1464), ADR(gc_DbmTranslation_en_Text1465), ADR(gc_DbmTranslation_en_Text1466), ADR(gc_DbmTranslation_en_Text1467), ADR(gc_DbmTranslation_en_Text1468), ADR(gc_DbmTranslation_en_Text1469), ADR(gc_DbmTranslation_en_Text1470), ADR(gc_DbmTranslation_en_Text1471), ADR(gc_DbmTranslation_en_Text1472), ADR(gc_DbmTranslation_en_Text1473), ADR(gc_DbmTranslation_en_Text1474), ADR(gc_DbmTranslation_en_Text1475), ADR(gc_DbmTranslation_en_Text1476), ADR(gc_DbmTranslation_en_Text1477), ADR(gc_DbmTranslation_en_Text1478), ADR(gc_DbmTranslation_en_Text1479), ADR(gc_DbmTranslation_en_Text1480), ADR(gc_DbmTranslation_en_Text1481), ADR(gc_DbmTranslation_en_Text1482), ADR(gc_DbmTranslation_en_Text1483), ADR(gc_DbmTranslation_en_Text1484), ADR(gc_DbmTranslation_en_Text1485), ADR(gc_DbmTranslation_en_Text1486), ADR(gc_DbmTranslation_en_Text1487), ADR(gc_DbmTranslation_en_Text1488), ADR(gc_DbmTranslation_en_Text1489), ADR(gc_DbmTranslation_en_Text1490), ADR(gc_DbmTranslation_en_Text1491), ADR(gc_DbmTranslation_en_Text1492), ADR(gc_DbmTranslation_en_Text1493), ADR(gc_DbmTranslation_en_Text1494), ADR(gc_DbmTranslation_en_Text1495), ADR(gc_DbmTranslation_en_Text1496), ADR(gc_DbmTranslation_en_Text1497), ADR(gc_DbmTranslation_en_Text1498), ADR(gc_DbmTranslation_en_Text1499), ADR(gc_DbmTranslation_en_Text1500), ADR(gc_DbmTranslation_en_Text1501), ADR(gc_DbmTranslation_en_Text1502), ADR(gc_DbmTranslation_en_Text1503), ADR(gc_DbmTranslation_en_Text1504), ADR(gc_DbmTranslation_en_Text1505), ADR(gc_DbmTranslation_en_Text1506), ADR(gc_DbmTranslation_en_Text1507), ADR(gc_DbmTranslation_en_Text1508), ADR(gc_DbmTranslation_en_Text1509), ADR(gc_DbmTranslation_en_Text1510), ADR(gc_DbmTranslation_en_Text1511), ADR(gc_DbmTranslation_en_Text1512), ADR(gc_DbmTranslation_en_Text1513), ADR(gc_DbmTranslation_en_Text1514), ADR(gc_DbmTranslation_en_Text1515), ADR(gc_DbmTranslation_en_Text1516), ADR(gc_DbmTranslation_en_Text1517), ADR(gc_DbmTranslation_en_Text1518), ADR(gc_DbmTranslation_en_Text1519), ADR(gc_DbmTranslation_en_Text1520), ADR(gc_DbmTranslation_en_Text1521), ADR(gc_DbmTranslation_en_Text1522), ADR(gc_DbmTranslation_en_Text1523), ADR(gc_DbmTranslation_en_Text1524), ADR(gc_DbmTranslation_en_Text1525), ADR(gc_DbmTranslation_en_Text1526), ADR(gc_DbmTranslation_en_Text1527), ADR(gc_DbmTranslation_en_Text1528), ADR(gc_DbmTranslation_en_Text1529), ADR(gc_DbmTranslation_en_Text1530), ADR(gc_DbmTranslation_en_Text1531), ADR(gc_DbmTranslation_en_Text1532), ADR(gc_DbmTranslation_en_Text1533), ADR(gc_DbmTranslation_en_Text1534), ADR(gc_DbmTranslation_en_Text1535), ADR(gc_DbmTranslation_en_Text1536), ADR(gc_DbmTranslation_en_Text1537), ADR(gc_DbmTranslation_en_Text1538), ADR(gc_DbmTranslation_en_Text1539), ADR(gc_DbmTranslation_en_Text1540), ADR(gc_DbmTranslation_en_Text1541), ADR(gc_DbmTranslation_en_Text1542), ADR(gc_DbmTranslation_en_Text1543), ADR(gc_DbmTranslation_en_Text1544), ADR(gc_DbmTranslation_en_Text1545), ADR(gc_DbmTranslation_en_Text1546), ADR(gc_DbmTranslation_en_Text1547), ADR(gc_DbmTranslation_en_Text1548), ADR(gc_DbmTranslation_en_Text1549), ADR(gc_DbmTranslation_en_Text1550), ADR(gc_DbmTranslation_en_Text1551), ADR(gc_DbmTranslation_en_Text1552), ADR(gc_DbmTranslation_en_Text1553), ADR(gc_DbmTranslation_en_Text1554), ADR(gc_DbmTranslation_en_Text1555), ADR(gc_DbmTranslation_en_Text1556), ADR(gc_DbmTranslation_en_Text1557), ADR(gc_DbmTranslation_en_Text1558), ADR(gc_DbmTranslation_en_Text1559), ADR(gc_DbmTranslation_en_Text1560), ADR(gc_DbmTranslation_en_Text1561), ADR(gc_DbmTranslation_en_Text1562), ADR(gc_DbmTranslation_en_Text1563), ADR(gc_DbmTranslation_en_Text1564), ADR(gc_DbmTranslation_en_Text1565), ADR(gc_DbmTranslation_en_Text1566), ADR(gc_DbmTranslation_en_Text1567), ADR(gc_DbmTranslation_en_Text1568), ADR(gc_DbmTranslation_en_Text1569), ADR(gc_DbmTranslation_en_Text1570), ADR(gc_DbmTranslation_en_Text1571), ADR(gc_DbmTranslation_en_Text1572), ADR(gc_DbmTranslation_en_Text1573), ADR(gc_DbmTranslation_en_Text1574), ADR(gc_DbmTranslation_en_Text1575), ADR(gc_DbmTranslation_en_Text1576), ADR(gc_DbmTranslation_en_Text1577), ADR(gc_DbmTranslation_en_Text1578), ADR(gc_DbmTranslation_en_Text1579), ADR(gc_DbmTranslation_en_Text1580), ADR(gc_DbmTranslation_en_Text1581), ADR(gc_DbmTranslation_en_Text1582), ADR(gc_DbmTranslation_en_Text1583), ADR(gc_DbmTranslation_en_Text1584), ADR(gc_DbmTranslation_en_Text1585), ADR(gc_DbmTranslation_en_Text1586), ADR(gc_DbmTranslation_en_Text1587), ADR(gc_DbmTranslation_en_Text1588), ADR(gc_DbmTranslation_en_Text1589), ADR(gc_DbmTranslation_en_Text1590), ADR(gc_DbmTranslation_en_Text1591), ADR(gc_DbmTranslation_en_Text1592), ADR(gc_DbmTranslation_en_Text1593), ADR(gc_DbmTranslation_en_Text1594), ADR(gc_DbmTranslation_en_Text1595), ADR(gc_DbmTranslation_en_Text1596), ADR(gc_DbmTranslation_en_Text1597), ADR(gc_DbmTranslation_en_Text1598), ADR(gc_DbmTranslation_en_Text1599), ADR(gc_DbmTranslation_en_Text1600), ADR(gc_DbmTranslation_en_Text1601), ADR(gc_DbmTranslation_en_Text1602), ADR(gc_DbmTranslation_en_Text1603), ADR(gc_DbmTranslation_en_Text1604), ADR(gc_DbmTranslation_en_Text1605), ADR(gc_DbmTranslation_en_Text1606), ADR(gc_DbmTranslation_en_Text1607), ADR(gc_DbmTranslation_en_Text1608), ADR(gc_DbmTranslation_en_Text1609), ADR(gc_DbmTranslation_en_Text1610), ADR(gc_DbmTranslation_en_Text1611), ADR(gc_DbmTranslation_en_Text1612), ADR(gc_DbmTranslation_en_Text1613), ADR(gc_DbmTranslation_en_Text1614), ADR(gc_DbmTranslation_en_Text1615), ADR(gc_DbmTranslation_en_Text1616), ADR(gc_DbmTranslation_en_Text1617), ADR(gc_DbmTranslation_en_Text1618), ADR(gc_DbmTranslation_en_Text1619), ADR(gc_DbmTranslation_en_Text1620), ADR(gc_DbmTranslation_en_Text1621), ADR(gc_DbmTranslation_en_Text1622), ADR(gc_DbmTranslation_en_Text1623), ADR(gc_DbmTranslation_en_Text1624), ADR(gc_DbmTranslation_en_Text1625), ADR(gc_DbmTranslation_en_Text1626), ADR(gc_DbmTranslation_en_Text1627), ADR(gc_DbmTranslation_en_Text1628), ADR(gc_DbmTranslation_en_Text1629), ADR(gc_DbmTranslation_en_Text1630), ADR(gc_DbmTranslation_en_Text1631), ADR(gc_DbmTranslation_en_Text1632), ADR(gc_DbmTranslation_en_Text1633), ADR(gc_DbmTranslation_en_Text1634), ADR(gc_DbmTranslation_en_Text1635), ADR(gc_DbmTranslation_en_Text1636), ADR(gc_DbmTranslation_en_Text1637), ADR(gc_DbmTranslation_en_Text1638), ADR(gc_DbmTranslation_en_Text1639), ADR(gc_DbmTranslation_en_Text1640), ADR(gc_DbmTranslation_en_Text1641), ADR(gc_DbmTranslation_en_Text1642), ADR(gc_DbmTranslation_en_Text1643), ADR(gc_DbmTranslation_en_Text1644), ADR(gc_DbmTranslation_en_Text1645), ADR(gc_DbmTranslation_en_Text1646), ADR(gc_DbmTranslation_en_Text1647), ADR(gc_DbmTranslation_en_Text1648), ADR(gc_DbmTranslation_en_Text1649), ADR(gc_DbmTranslation_en_Text1650), ADR(gc_DbmTranslation_en_Text1651), ADR(gc_DbmTranslation_en_Text1652), ADR(gc_DbmTranslation_en_Text1653), ADR(gc_DbmTranslation_en_Text1654), ADR(gc_DbmTranslation_en_Text1655), ADR(gc_DbmTranslation_en_Text1656), ADR(gc_DbmTranslation_en_Text1657), ADR(gc_DbmTranslation_en_Text1658), ADR(gc_DbmTranslation_en_Text1659), ADR(gc_DbmTranslation_en_Text1660), ADR(gc_DbmTranslation_en_Text1661), ADR(gc_DbmTranslation_en_Text1662), ADR(gc_DbmTranslation_en_Text1663), ADR(gc_DbmTranslation_en_Text1664), ADR(gc_DbmTranslation_en_Text1665), ADR(gc_DbmTranslation_en_Text1666), ADR(gc_DbmTranslation_en_Text1667), ADR(gc_DbmTranslation_en_Text1668), ADR(gc_DbmTranslation_en_Text1669), ADR(gc_DbmTranslation_en_Text1670), ADR(gc_DbmTranslation_en_Text1671), ADR(gc_DbmTranslation_en_Text1672), ADR(gc_DbmTranslation_en_Text1673), ADR(gc_DbmTranslation_en_Text1674), ADR(gc_DbmTranslation_en_Text1675), ADR(gc_DbmTranslation_en_Text1676), ADR(gc_DbmTranslation_en_Text1677), ADR(gc_DbmTranslation_en_Text1678), ADR(gc_DbmTranslation_en_Text1679), ADR(gc_DbmTranslation_en_Text1680), ADR(gc_DbmTranslation_en_Text1681), ADR(gc_DbmTranslation_en_Text1682), ADR(gc_DbmTranslation_en_Text1683), ADR(gc_DbmTranslation_en_Text1684), ADR(gc_DbmTranslation_en_Text1685), ADR(gc_DbmTranslation_en_Text1686), ADR(gc_DbmTranslation_en_Text1687), ADR(gc_DbmTranslation_en_Text1688), ADR(gc_DbmTranslation_en_Text1689), ADR(gc_DbmTranslation_en_Text1690), ADR(gc_DbmTranslation_en_Text1691), ADR(gc_DbmTranslation_en_Text1692), ADR(gc_DbmTranslation_en_Text1693), ADR(gc_DbmTranslation_en_Text1694), ADR(gc_DbmTranslation_en_Text1695), ADR(gc_DbmTranslation_en_Text1696), ADR(gc_DbmTranslation_en_Text1697), ADR(gc_DbmTranslation_en_Text1698), ADR(gc_DbmTranslation_en_Text1699), ADR(gc_DbmTranslation_en_Text1700), ADR(gc_DbmTranslation_en_Text1701), ADR(gc_DbmTranslation_en_Text1702), ADR(gc_DbmTranslation_en_Text1703), ADR(gc_DbmTranslation_en_Text1704), ADR(gc_DbmTranslation_en_Text1705), ADR(gc_DbmTranslation_en_Text1706), ADR(gc_DbmTranslation_en_Text1707), ADR(gc_DbmTranslation_en_Text1708), ADR(gc_DbmTranslation_en_Text1709), ADR(gc_DbmTranslation_en_Text1710), ADR(gc_DbmTranslation_en_Text1711), ADR(gc_DbmTranslation_en_Text1712), ADR(gc_DbmTranslation_en_Text1713), ADR(gc_DbmTranslation_en_Text1714), ADR(gc_DbmTranslation_en_Text1715), ADR(gc_DbmTranslation_en_Text1716), ADR(gc_DbmTranslation_en_Text1717), ADR(gc_DbmTranslation_en_Text1718), ADR(gc_DbmTranslation_en_Text1719), ADR(gc_DbmTranslation_en_Text1720), ADR(gc_DbmTranslation_en_Text1721), ADR(gc_DbmTranslation_en_Text1722), ADR(gc_DbmTranslation_en_Text1723), ADR(gc_DbmTranslation_en_Text1724), ADR(gc_DbmTranslation_en_Text1725), ADR(gc_DbmTranslation_en_Text1726), ADR(gc_DbmTranslation_en_Text1727), ADR(gc_DbmTranslation_en_Text1728), ADR(gc_DbmTranslation_en_Text1729), ADR(gc_DbmTranslation_en_Text1730), ADR(gc_DbmTranslation_en_Text1731), ADR(gc_DbmTranslation_en_Text1732), ADR(gc_DbmTranslation_en_Text1733), ADR(gc_DbmTranslation_en_Text1734), ADR(gc_DbmTranslation_en_Text1735), ADR(gc_DbmTranslation_en_Text1736), ADR(gc_DbmTranslation_en_Text1737), ADR(gc_DbmTranslation_en_Text1738), ADR(gc_DbmTranslation_en_Text1739), ADR(gc_DbmTranslation_en_Text1740), ADR(gc_DbmTranslation_en_Text1741), ADR(gc_DbmTranslation_en_Text1742), ADR(gc_DbmTranslation_en_Text1743), ADR(gc_DbmTranslation_en_Text1744), ADR(gc_DbmTranslation_en_Text1745), ADR(gc_DbmTranslation_en_Text1746), ADR(gc_DbmTranslation_en_Text1747), ADR(gc_DbmTranslation_en_Text1748), ADR(gc_DbmTranslation_en_Text1749), ADR(gc_DbmTranslation_en_Text1750), ADR(gc_DbmTranslation_en_Text1751), ADR(gc_DbmTranslation_en_Text1752), ADR(gc_DbmTranslation_en_Text1753), ADR(gc_DbmTranslation_en_Text1754), ADR(gc_DbmTranslation_en_Text1755), ADR(gc_DbmTranslation_en_Text1756), ADR(gc_DbmTranslation_en_Text1757), ADR(gc_DbmTranslation_en_Text1758), ADR(gc_DbmTranslation_en_Text1759), ADR(gc_DbmTranslation_en_Text1760), ADR(gc_DbmTranslation_en_Text1761), ADR(gc_DbmTranslation_en_Text1762), ADR(gc_DbmTranslation_en_Text1763), ADR(gc_DbmTranslation_en_Text1764), ADR(gc_DbmTranslation_en_Text1765), ADR(gc_DbmTranslation_en_Text1766), ADR(gc_DbmTranslation_en_Text1767), ADR(gc_DbmTranslation_en_Text1768), ADR(gc_DbmTranslation_en_Text1769), ADR(gc_DbmTranslation_en_Text1770), ADR(gc_DbmTranslation_en_Text1771), ADR(gc_DbmTranslation_en_Text1772), ADR(gc_DbmTranslation_en_Text1773), ADR(gc_DbmTranslation_en_Text1774), ADR(gc_DbmTranslation_en_Text1775), ADR(gc_DbmTranslation_en_Text1776), ADR(gc_DbmTranslation_en_Text1777), ADR(gc_DbmTranslation_en_Text1778), ADR(gc_DbmTranslation_en_Text1779), ADR(gc_DbmTranslation_en_Text1780), ADR(gc_DbmTranslation_en_Text1781), ADR(gc_DbmTranslation_en_Text1782), ADR(gc_DbmTranslation_en_Text1783), ADR(gc_DbmTranslation_en_Text1784), ADR(gc_DbmTranslation_en_Text1785), ADR(gc_DbmTranslation_en_Text1786), ADR(gc_DbmTranslation_en_Text1787), ADR(gc_DbmTranslation_en_Text1788), ADR(gc_DbmTranslation_en_Text1789), ADR(gc_DbmTranslation_en_Text1790), ADR(gc_DbmTranslation_en_Text1791), ADR(gc_DbmTranslation_en_Text1792), ADR(gc_DbmTranslation_en_Text1793), ADR(gc_DbmTranslation_en_Text1794), ADR(gc_DbmTranslation_en_Text1795), ADR(gc_DbmTranslation_en_Text1796), ADR(gc_DbmTranslation_en_Text1797), ADR(gc_DbmTranslation_en_Text1798), ADR(gc_DbmTranslation_en_Text1799), ADR(gc_DbmTranslation_en_Text1800), ADR(gc_DbmTranslation_en_Text1801), ADR(gc_DbmTranslation_en_Text1802), ADR(gc_DbmTranslation_en_Text1803), ADR(gc_DbmTranslation_en_Text1804), ADR(gc_DbmTranslation_en_Text1805), ADR(gc_DbmTranslation_en_Text1806), ADR(gc_DbmTranslation_en_Text1807), ADR(gc_DbmTranslation_en_Text1808), ADR(gc_DbmTranslation_en_Text1809), ADR(gc_DbmTranslation_en_Text1810), ADR(gc_DbmTranslation_en_Text1811), ADR(gc_DbmTranslation_en_Text1812), ADR(gc_DbmTranslation_en_Text1813), ADR(gc_DbmTranslation_en_Text1814), ADR(gc_DbmTranslation_en_Text1815), ADR(gc_DbmTranslation_en_Text1816), ADR(gc_DbmTranslation_en_Text1817), ADR(gc_DbmTranslation_en_Text1818), ADR(gc_DbmTranslation_en_Text1819), ADR(gc_DbmTranslation_en_Text1820), ADR(gc_DbmTranslation_en_Text1821), ADR(gc_DbmTranslation_en_Text1822), ADR(gc_DbmTranslation_en_Text1823), ADR(gc_DbmTranslation_en_Text1824), ADR(gc_DbmTranslation_en_Text1825), ADR(gc_DbmTranslation_en_Text1826), ADR(gc_DbmTranslation_en_Text1827), ADR(gc_DbmTranslation_en_Text1828), ADR(gc_DbmTranslation_en_Text1829), ADR(gc_DbmTranslation_en_Text1830), ADR(gc_DbmTranslation_en_Text1831), ADR(gc_DbmTranslation_en_Text1832), ADR(gc_DbmTranslation_en_Text1833), ADR(gc_DbmTranslation_en_Text1834), ADR(gc_DbmTranslation_en_Text1835), ADR(gc_DbmTranslation_en_Text1836), ADR(gc_DbmTranslation_en_Text1837), ADR(gc_DbmTranslation_en_Text1838), ADR(gc_DbmTranslation_en_Text1839), ADR(gc_DbmTranslation_en_Text1840), ADR(gc_DbmTranslation_en_Text1841), ADR(gc_DbmTranslation_en_Text1842), ADR(gc_DbmTranslation_en_Text1843), ADR(gc_DbmTranslation_en_Text1844), ADR(gc_DbmTranslation_en_Text1845), ADR(gc_DbmTranslation_en_Text1846), ADR(gc_DbmTranslation_en_Text1847), ADR(gc_DbmTranslation_en_Text1848), ADR(gc_DbmTranslation_en_Text1849), ADR(gc_DbmTranslation_en_Text1850), ADR(gc_DbmTranslation_en_Text1851), ADR(gc_DbmTranslation_en_Text1852), ADR(gc_DbmTranslation_en_Text1853), ADR(gc_DbmTranslation_en_Text1854), ADR(gc_DbmTranslation_en_Text1855), ADR(gc_DbmTranslation_en_Text1856), ADR(gc_DbmTranslation_en_Text1857), ADR(gc_DbmTranslation_en_Text1858), ADR(gc_DbmTranslation_en_Text1859), ADR(gc_DbmTranslation_en_Text1860), ADR(gc_DbmTranslation_en_Text1861), ADR(gc_DbmTranslation_en_Text1862), ADR(gc_DbmTranslation_en_Text1863), ADR(gc_DbmTranslation_en_Text1864), ADR(gc_DbmTranslation_en_Text1865), ADR(gc_DbmTranslation_en_Text1866), ADR(gc_DbmTranslation_en_Text1867), ADR(gc_DbmTranslation_en_Text1868), ADR(gc_DbmTranslation_en_Text1869), ADR(gc_DbmTranslation_en_Text1870), ADR(gc_DbmTranslation_en_Text1871), ADR(gc_DbmTranslation_en_Text1872), ADR(gc_DbmTranslation_en_Text1873), ADR(gc_DbmTranslation_en_Text1874), ADR(gc_DbmTranslation_en_Text1875), ADR(gc_DbmTranslation_en_Text1876), ADR(gc_DbmTranslation_en_Text1877), ADR(gc_DbmTranslation_en_Text1878), ADR(gc_DbmTranslation_en_Text1879), ADR(gc_DbmTranslation_en_Text1880), ADR(gc_DbmTranslation_en_Text1881), ADR(gc_DbmTranslation_en_Text1882), ADR(gc_DbmTranslation_en_Text1883), ADR(gc_DbmTranslation_en_Text1884), ADR(gc_DbmTranslation_en_Text1885), ADR(gc_DbmTranslation_en_Text1886), ADR(gc_DbmTranslation_en_Text1887), ADR(gc_DbmTranslation_en_Text1888), ADR(gc_DbmTranslation_en_Text1889), ADR(gc_DbmTranslation_en_Text1890), ADR(gc_DbmTranslation_en_Text1891), ADR(gc_DbmTranslation_en_Text1892), ADR(gc_DbmTranslation_en_Text1893), ADR(gc_DbmTranslation_en_Text1894), ADR(gc_DbmTranslation_en_Text1895), ADR(gc_DbmTranslation_en_Text1896), ADR(gc_DbmTranslation_en_Text1897), ADR(gc_DbmTranslation_en_Text1898), ADR(gc_DbmTranslation_en_Text1899), ADR(gc_DbmTranslation_en_Text1900), ADR(gc_DbmTranslation_en_Text1901), ADR(gc_DbmTranslation_en_Text1902), ADR(gc_DbmTranslation_en_Text1903), ADR(gc_DbmTranslation_en_Text1904), ADR(gc_DbmTranslation_en_Text1905), ADR(gc_DbmTranslation_en_Text1906), ADR(gc_DbmTranslation_en_Text1907), ADR(gc_DbmTranslation_en_Text1908), ADR(gc_DbmTranslation_en_Text1909), ADR(gc_DbmTranslation_en_Text1910), ADR(gc_DbmTranslation_en_Text1911), ADR(gc_DbmTranslation_en_Text1912), ADR(gc_DbmTranslation_en_Text1913), ADR(gc_DbmTranslation_en_Text1914), ADR(gc_DbmTranslation_en_Text1915), ADR(gc_DbmTranslation_en_Text1916), ADR(gc_DbmTranslation_en_Text1917), ADR(gc_DbmTranslation_en_Text1918), ADR(gc_DbmTranslation_en_Text1919), ADR(gc_DbmTranslation_en_Text1920), ADR(gc_DbmTranslation_en_Text1921), ADR(gc_DbmTranslation_en_Text1922), ADR(gc_DbmTranslation_en_Text1923), ADR(gc_DbmTranslation_en_Text1924), ADR(gc_DbmTranslation_en_Text1925), ADR(gc_DbmTranslation_en_Text1926), ADR(gc_DbmTranslation_en_Text1927), ADR(gc_DbmTranslation_en_Text1928), ADR(gc_DbmTranslation_en_Text1929), ADR(gc_DbmTranslation_en_Text1930), ADR(gc_DbmTranslation_en_Text1931), ADR(gc_DbmTranslation_en_Text1932), ADR(gc_DbmTranslation_en_Text1933), ADR(gc_DbmTranslation_en_Text1934), ADR(gc_DbmTranslation_en_Text1935), ADR(gc_DbmTranslation_en_Text1936), ADR(gc_DbmTranslation_en_Text1937), ADR(gc_DbmTranslation_en_Text1938), ADR(gc_DbmTranslation_en_Text1939), ADR(gc_DbmTranslation_en_Text1940), ADR(gc_DbmTranslation_en_Text1941), ADR(gc_DbmTranslation_en_Text1942), ADR(gc_DbmTranslation_en_Text1943), ADR(gc_DbmTranslation_en_Text1944), ADR(gc_DbmTranslation_en_Text1945), ADR(gc_DbmTranslation_en_Text1946), ADR(gc_DbmTranslation_en_Text1947), ADR(gc_DbmTranslation_en_Text1948), ADR(gc_DbmTranslation_en_Text1949), ADR(gc_DbmTranslation_en_Text1950), ADR(gc_DbmTranslation_en_Text1951), ADR(gc_DbmTranslation_en_Text1952), ADR(gc_DbmTranslation_en_Text1953), ADR(gc_DbmTranslation_en_Text1954), ADR(gc_DbmTranslation_en_Text1955), ADR(gc_DbmTranslation_en_Text1956), ADR(gc_DbmTranslation_en_Text1957), ADR(gc_DbmTranslation_en_Text1958), ADR(gc_DbmTranslation_en_Text1959), ADR(gc_DbmTranslation_en_Text1960), ADR(gc_DbmTranslation_en_Text1961), ADR(gc_DbmTranslation_en_Text1962), ADR(gc_DbmTranslation_en_Text1963), ADR(gc_DbmTranslation_en_Text1964), ADR(gc_DbmTranslation_en_Text1965), ADR(gc_DbmTranslation_en_Text1966), ADR(gc_DbmTranslation_en_Text1967), ADR(gc_DbmTranslation_en_Text1968), ADR(gc_DbmTranslation_en_Text1969), ADR(gc_DbmTranslation_en_Text1970), ADR(gc_DbmTranslation_en_Text1971), ADR(gc_DbmTranslation_en_Text1972), ADR(gc_DbmTranslation_en_Text1973), ADR(gc_DbmTranslation_en_Text1974), ADR(gc_DbmTranslation_en_Text1975), ADR(gc_DbmTranslation_en_Text1976), ADR(gc_DbmTranslation_en_Text1977), ADR(gc_DbmTranslation_en_Text1978), ADR(gc_DbmTranslation_en_Text1979), ADR(gc_DbmTranslation_en_Text1980), ADR(gc_DbmTranslation_en_Text1981), ADR(gc_DbmTranslation_en_Text1982), ADR(gc_DbmTranslation_en_Text1983), ADR(gc_DbmTranslation_en_Text1984), ADR(gc_DbmTranslation_en_Text1985), ADR(gc_DbmTranslation_en_Text1986), ADR(gc_DbmTranslation_en_Text1987), ADR(gc_DbmTranslation_en_Text1988), ADR(gc_DbmTranslation_en_Text1989), ADR(gc_DbmTranslation_en_Text1990), ADR(gc_DbmTranslation_en_Text1991), ADR(gc_DbmTranslation_en_Text1992), ADR(gc_DbmTranslation_en_Text1993), ADR(gc_DbmTranslation_en_Text1994), ADR(gc_DbmTranslation_en_Text1995), ADR(gc_DbmTranslation_en_Text1996), ADR(gc_DbmTranslation_en_Text1997), ADR(gc_DbmTranslation_en_Text1998), ADR(gc_DbmTranslation_en_Text1999), ADR(gc_DbmTranslation_en_Text2000), ADR(gc_DbmTranslation_en_Text2001), ADR(gc_DbmTranslation_en_Text2002), ADR(gc_DbmTranslation_en_Text2003), ADR(gc_DbmTranslation_en_Text2004), ADR(gc_DbmTranslation_en_Text2005), ADR(gc_DbmTranslation_en_Text2006), ADR(gc_DbmTranslation_en_Text2007), ADR(gc_DbmTranslation_en_Text2008), ADR(gc_DbmTranslation_en_Text2009), ADR(gc_DbmTranslation_en_Text2010), ADR(gc_DbmTranslation_en_Text2011), ADR(gc_DbmTranslation_en_Text2012), ADR(gc_DbmTranslation_en_Text2013), ADR(gc_DbmTranslation_en_Text2014), ADR(gc_DbmTranslation_en_Text2015), ADR(gc_DbmTranslation_en_Text2016), ADR(gc_DbmTranslation_en_Text2017), ADR(gc_DbmTranslation_en_Text2018), ADR(gc_DbmTranslation_en_Text2019), ADR(gc_DbmTranslation_en_Text2020), ADR(gc_DbmTranslation_en_Text2021), ADR(gc_DbmTranslation_en_Text2022), ADR(gc_DbmTranslation_en_Text2023), ADR(gc_DbmTranslation_en_Text2024), ADR(gc_DbmTranslation_en_Text2025), ADR(gc_DbmTranslation_en_Text2026), ADR(gc_DbmTranslation_en_Text2027), ADR(gc_DbmTranslation_en_Text2028), ADR(gc_DbmTranslation_en_Text2029), ADR(gc_DbmTranslation_en_Text2030), ADR(gc_DbmTranslation_en_Text2031), ADR(gc_DbmTranslation_en_Text2032), ADR(gc_DbmTranslation_en_Text2033), ADR(gc_DbmTranslation_en_Text2034), ADR(gc_DbmTranslation_en_Text2035), ADR(gc_DbmTranslation_en_Text2036), ADR(gc_DbmTranslation_en_Text2037), ADR(gc_DbmTranslation_en_Text2038), ADR(gc_DbmTranslation_en_Text2039), ADR(gc_DbmTranslation_en_Text2040), ADR(gc_DbmTranslation_en_Text2041), ADR(gc_DbmTranslation_en_Text2042), ADR(gc_DbmTranslation_en_Text2043), ADR(gc_DbmTranslation_en_Text2044), ADR(gc_DbmTranslation_en_Text2045), ADR(gc_DbmTranslation_en_Text2046), ADR(gc_DbmTranslation_en_Text2047), ADR(gc_DbmTranslation_en_Text2048), ADR(gc_DbmTranslation_en_Text2049), ADR(gc_DbmTranslation_en_Text2050), ADR(gc_DbmTranslation_en_Text2051), ADR(gc_DbmTranslation_en_Text2052), ADR(gc_DbmTranslation_en_Text2053), ADR(gc_DbmTranslation_en_Text2054), ADR(gc_DbmTranslation_en_Text2055), ADR(gc_DbmTranslation_en_Text2056), ADR(gc_DbmTranslation_en_Text2057), ADR(gc_DbmTranslation_en_Text2058), ADR(gc_DbmTranslation_en_Text2059), ADR(gc_DbmTranslation_en_Text2060), ADR(gc_DbmTranslation_en_Text2061), ADR(gc_DbmTranslation_en_Text2062), ADR(gc_DbmTranslation_en_Text2063), ADR(gc_DbmTranslation_en_Text2064), ADR(gc_DbmTranslation_en_Text2065), ADR(gc_DbmTranslation_en_Text2066), ADR(gc_DbmTranslation_en_Text2067), ADR(gc_DbmTranslation_en_Text2068), ADR(gc_DbmTranslation_en_Text2069), ADR(gc_DbmTranslation_en_Text2070), ADR(gc_DbmTranslation_en_Text2071), ADR(gc_DbmTranslation_en_Text2072), ADR(gc_DbmTranslation_en_Text2073), ADR(gc_DbmTranslation_en_Text2074), ADR(gc_DbmTranslation_en_Text2075), ADR(gc_DbmTranslation_en_Text2076), ADR(gc_DbmTranslation_en_Text2077), ADR(gc_DbmTranslation_en_Text2078), ADR(gc_DbmTranslation_en_Text2079), ADR(gc_DbmTranslation_en_Text2080), ADR(gc_DbmTranslation_en_Text2081), ADR(gc_DbmTranslation_en_Text2082), ADR(gc_DbmTranslation_en_Text2083), ADR(gc_DbmTranslation_en_Text2084), ADR(gc_DbmTranslation_en_Text2085), ADR(gc_DbmTranslation_en_Text2086), ADR(gc_DbmTranslation_en_Text2087), ADR(gc_DbmTranslation_en_Text2088), ADR(gc_DbmTranslation_en_Text2089), ADR(gc_DbmTranslation_en_Text2090), ADR(gc_DbmTranslation_en_Text2091), ADR(gc_DbmTranslation_en_Text2092), ADR(gc_DbmTranslation_en_Text2093), ADR(gc_DbmTranslation_en_Text2094), ADR(gc_DbmTranslation_en_Text2095), ADR(gc_DbmTranslation_en_Text2096), ADR(gc_DbmTranslation_en_Text2097), ADR(gc_DbmTranslation_en_Text2098), ADR(gc_DbmTranslation_en_Text2099), ADR(gc_DbmTranslation_en_Text2100), ADR(gc_DbmTranslation_en_Text2101), ADR(gc_DbmTranslation_en_Text2102), ADR(gc_DbmTranslation_en_Text2103), ADR(gc_DbmTranslation_en_Text2104), ADR(gc_DbmTranslation_en_Text2105), ADR(gc_DbmTranslation_en_Text2106), ADR(gc_DbmTranslation_en_Text2107), ADR(gc_DbmTranslation_en_Text2108), ADR(gc_DbmTranslation_en_Text2109), ADR(gc_DbmTranslation_en_Text2110), ADR(gc_DbmTranslation_en_Text2111), ADR(gc_DbmTranslation_en_Text2112), ADR(gc_DbmTranslation_en_Text2113), ADR(gc_DbmTranslation_en_Text2114), ADR(gc_DbmTranslation_en_Text2115), ADR(gc_DbmTranslation_en_Text2116), ADR(gc_DbmTranslation_en_Text2117), ADR(gc_DbmTranslation_en_Text2118), ADR(gc_DbmTranslation_en_Text2119), ADR(gc_DbmTranslation_en_Text2120), ADR(gc_DbmTranslation_en_Text2121), ADR(gc_DbmTranslation_en_Text2122), ADR(gc_DbmTranslation_en_Text2123), ADR(gc_DbmTranslation_en_Text2124), ADR(gc_DbmTranslation_en_Text2125), ADR(gc_DbmTranslation_en_Text2126), ADR(gc_DbmTranslation_en_Text2127), ADR(gc_DbmTranslation_en_Text2128), ADR(gc_DbmTranslation_en_Text2129), ADR(gc_DbmTranslation_en_Text2130), ADR(gc_DbmTranslation_en_Text2131), ADR(gc_DbmTranslation_en_Text2132), ADR(gc_DbmTranslation_en_Text2133), ADR(gc_DbmTranslation_en_Text2134), ADR(gc_DbmTranslation_en_Text2135), ADR(gc_DbmTranslation_en_Text2136), ADR(gc_DbmTranslation_en_Text2137), ADR(gc_DbmTranslation_en_Text2138), ADR(gc_DbmTranslation_en_Text2139), ADR(gc_DbmTranslation_en_Text2140), ADR(gc_DbmTranslation_en_Text2141), ADR(gc_DbmTranslation_en_Text2142), ADR(gc_DbmTranslation_en_Text2143), ADR(gc_DbmTranslation_en_Text2144), ADR(gc_DbmTranslation_en_Text2145), ADR(gc_DbmTranslation_en_Text2146), ADR(gc_DbmTranslation_en_Text2147), ADR(gc_DbmTranslation_en_Text2148), ADR(gc_DbmTranslation_en_Text2149), ADR(gc_DbmTranslation_en_Text2150), ADR(gc_DbmTranslation_en_Text2151), ADR(gc_DbmTranslation_en_Text2152), ADR(gc_DbmTranslation_en_Text2153), ADR(gc_DbmTranslation_en_Text2154), ADR(gc_DbmTranslation_en_Text2155), ADR(gc_DbmTranslation_en_Text2156), ADR(gc_DbmTranslation_en_Text2157), ADR(gc_DbmTranslation_en_Text2158), ADR(gc_DbmTranslation_en_Text2159), ADR(gc_DbmTranslation_en_Text2160), ADR(gc_DbmTranslation_en_Text2161), ADR(gc_DbmTranslation_en_Text2162), ADR(gc_DbmTranslation_en_Text2163), ADR(gc_DbmTranslation_en_Text2164), ADR(gc_DbmTranslation_en_Text2165), ADR(gc_DbmTranslation_en_Text2166), ADR(gc_DbmTranslation_en_Text2167), ADR(gc_DbmTranslation_en_Text2168), ADR(gc_DbmTranslation_en_Text2169), ADR(gc_DbmTranslation_en_Text2170), ADR(gc_DbmTranslation_en_Text2171), ADR(gc_DbmTranslation_en_Text2172), ADR(gc_DbmTranslation_en_Text2173), ADR(gc_DbmTranslation_en_Text2174), ADR(gc_DbmTranslation_en_Text2175), ADR(gc_DbmTranslation_en_Text2176), ADR(gc_DbmTranslation_en_Text2177), ADR(gc_DbmTranslation_en_Text2178), ADR(gc_DbmTranslation_en_Text2179), ADR(gc_DbmTranslation_en_Text2180), ADR(gc_DbmTranslation_en_Text2181), ADR(gc_DbmTranslation_en_Text2182), ADR(gc_DbmTranslation_en_Text2183), ADR(gc_DbmTranslation_en_Text2184), ADR(gc_DbmTranslation_en_Text2185), ADR(gc_DbmTranslation_en_Text2186), ADR(gc_DbmTranslation_en_Text2187), ADR(gc_DbmTranslation_en_Text2188), ADR(gc_DbmTranslation_en_Text2189), ADR(gc_DbmTranslation_en_Text2190), ADR(gc_DbmTranslation_en_Text2191), ADR(gc_DbmTranslation_en_Text2192), ADR(gc_DbmTranslation_en_Text2193), ADR(gc_DbmTranslation_en_Text2194), ADR(gc_DbmTranslation_en_Text2195), ADR(gc_DbmTranslation_en_Text2196), ADR(gc_DbmTranslation_en_Text2197), ADR(gc_DbmTranslation_en_Text2198), ADR(gc_DbmTranslation_en_Text2199), ADR(gc_DbmTranslation_en_Text2200), ADR(gc_DbmTranslation_en_Text2201), ADR(gc_DbmTranslation_en_Text2202), ADR(gc_DbmTranslation_en_Text2203), ADR(gc_DbmTranslation_en_Text2204), ADR(gc_DbmTranslation_en_Text2205), ADR(gc_DbmTranslation_en_Text2206), ADR(gc_DbmTranslation_en_Text2207), ADR(gc_DbmTranslation_en_Text2208), ADR(gc_DbmTranslation_en_Text2209), ADR(gc_DbmTranslation_en_Text2210), ADR(gc_DbmTranslation_en_Text2211), ADR(gc_DbmTranslation_en_Text2212), ADR(gc_DbmTranslation_en_Text2213), ADR(gc_DbmTranslation_en_Text2214), ADR(gc_DbmTranslation_en_Text2215), ADR(gc_DbmTranslation_en_Text2216), ADR(gc_DbmTranslation_en_Text2217), ADR(gc_DbmTranslation_en_Text2218), ADR(gc_DbmTranslation_en_Text2219), ADR(gc_DbmTranslation_en_Text2220), ADR(gc_DbmTranslation_en_Text2221), ADR(gc_DbmTranslation_en_Text2222), ADR(gc_DbmTranslation_en_Text2223), ADR(gc_DbmTranslation_en_Text2224), ADR(gc_DbmTranslation_en_Text2225), ADR(gc_DbmTranslation_en_Text2226), ADR(gc_DbmTranslation_en_Text2227), ADR(gc_DbmTranslation_en_Text2228), ADR(gc_DbmTranslation_en_Text2229), ADR(gc_DbmTranslation_en_Text2230), ADR(gc_DbmTranslation_en_Text2231), ADR(gc_DbmTranslation_en_Text2232), ADR(gc_DbmTranslation_en_Text2233), ADR(gc_DbmTranslation_en_Text2234), ADR(gc_DbmTranslation_en_Text2235), ADR(gc_DbmTranslation_en_Text2236), ADR(gc_DbmTranslation_en_Text2237), ADR(gc_DbmTranslation_en_Text2238), ADR(gc_DbmTranslation_en_Text2239), ADR(gc_DbmTranslation_en_Text2240), ADR(gc_DbmTranslation_en_Text2241), ADR(gc_DbmTranslation_en_Text2242), ADR(gc_DbmTranslation_en_Text2243), ADR(gc_DbmTranslation_en_Text2244), ADR(gc_DbmTranslation_en_Text2245), ADR(gc_DbmTranslation_en_Text2246), ADR(gc_DbmTranslation_en_Text2247), ADR(gc_DbmTranslation_en_Text2248), ADR(gc_DbmTranslation_en_Text2249), ADR(gc_DbmTranslation_en_Text2250), ADR(gc_DbmTranslation_en_Text2251), ADR(gc_DbmTranslation_en_Text2252), ADR(gc_DbmTranslation_en_Text2253), ADR(gc_DbmTranslation_en_Text2254), ADR(gc_DbmTranslation_en_Text2255), ADR(gc_DbmTranslation_en_Text2256), ADR(gc_DbmTranslation_en_Text2257), ADR(gc_DbmTranslation_en_Text2258), ADR(gc_DbmTranslation_en_Text2259), ADR(gc_DbmTranslation_en_Text2260), ADR(gc_DbmTranslation_en_Text2261), ADR(gc_DbmTranslation_en_Text2262), ADR(gc_DbmTranslation_en_Text2263), ADR(gc_DbmTranslation_en_Text2264), ADR(gc_DbmTranslation_en_Text2265), ADR(gc_DbmTranslation_en_Text2266), ADR(gc_DbmTranslation_en_Text2267), ADR(gc_DbmTranslation_en_Text2268), ADR(gc_DbmTranslation_en_Text2269), ADR(gc_DbmTranslation_en_Text2270), ADR(gc_DbmTranslation_en_Text2271), ADR(gc_DbmTranslation_en_Text2272), ADR(gc_DbmTranslation_en_Text2273), ADR(gc_DbmTranslation_en_Text2274), ADR(gc_DbmTranslation_en_Text2275), ADR(gc_DbmTranslation_en_Text2276), ADR(gc_DbmTranslation_en_Text2277), ADR(gc_DbmTranslation_en_Text2278), ADR(gc_DbmTranslation_en_Text2279), ADR(gc_DbmTranslation_en_Text2280), ADR(gc_DbmTranslation_en_Text2281), ADR(gc_DbmTranslation_en_Text2282), ADR(gc_DbmTranslation_en_Text2283), ADR(gc_DbmTranslation_en_Text2284), ADR(gc_DbmTranslation_en_Text2285), ADR(gc_DbmTranslation_en_Text2286), ADR(gc_DbmTranslation_en_Text2287), ADR(gc_DbmTranslation_en_Text2288), ADR(gc_DbmTranslation_en_Text2289), ADR(gc_DbmTranslation_en_Text2290), ADR(gc_DbmTranslation_en_Text2291), ADR(gc_DbmTranslation_en_Text2292), ADR(gc_DbmTranslation_en_Text2293), ADR(gc_DbmTranslation_en_Text2294), ADR(gc_DbmTranslation_en_Text2295), ADR(gc_DbmTranslation_en_Text2296), ADR(gc_DbmTranslation_en_Text2297), ADR(gc_DbmTranslation_en_Text2298), ADR(gc_DbmTranslation_en_Text2299), ADR(gc_DbmTranslation_en_Text2300), ADR(gc_DbmTranslation_en_Text2301), ADR(gc_DbmTranslation_en_Text2302), ADR(gc_DbmTranslation_en_Text2303), ADR(gc_DbmTranslation_en_Text2304), ADR(gc_DbmTranslation_en_Text2305), ADR(gc_DbmTranslation_en_Text2306), ADR(gc_DbmTranslation_en_Text2307), ADR(gc_DbmTranslation_en_Text2308), ADR(gc_DbmTranslation_en_Text2309), ADR(gc_DbmTranslation_en_Text2310), ADR(gc_DbmTranslation_en_Text2311), ADR(gc_DbmTranslation_en_Text2312), ADR(gc_DbmTranslation_en_Text2313), ADR(gc_DbmTranslation_en_Text2314), ADR(gc_DbmTranslation_en_Text2315), ADR(gc_DbmTranslation_en_Text2316), ADR(gc_DbmTranslation_en_Text2317), ADR(gc_DbmTranslation_en_Text2318), ADR(gc_DbmTranslation_en_Text2319), ADR(gc_DbmTranslation_en_Text2320), ADR(gc_DbmTranslation_en_Text2321), ADR(gc_DbmTranslation_en_Text2322), ADR(gc_DbmTranslation_en_Text2323), ADR(gc_DbmTranslation_en_Text2324), ADR(gc_DbmTranslation_en_Text2325), ADR(gc_DbmTranslation_en_Text2326), ADR(gc_DbmTranslation_en_Text2327), ADR(gc_DbmTranslation_en_Text2328), ADR(gc_DbmTranslation_en_Text2329), ADR(gc_DbmTranslation_en_Text2330), ADR(gc_DbmTranslation_en_Text2331), ADR(gc_DbmTranslation_en_Text2332), ADR(gc_DbmTranslation_en_Text2333), ADR(gc_DbmTranslation_en_Text2334), ADR(gc_DbmTranslation_en_Text2335), ADR(gc_DbmTranslation_en_Text2336), ADR(gc_DbmTranslation_en_Text2337), ADR(gc_DbmTranslation_en_Text2338), ADR(gc_DbmTranslation_en_Text2339), ADR(gc_DbmTranslation_en_Text2340), ADR(gc_DbmTranslation_en_Text2341), ADR(gc_DbmTranslation_en_Text2342), ADR(gc_DbmTranslation_en_Text2343), ADR(gc_DbmTranslation_en_Text2344), ADR(gc_DbmTranslation_en_Text2345), ADR(gc_DbmTranslation_en_Text2346), ADR(gc_DbmTranslation_en_Text2347), ADR(gc_DbmTranslation_en_Text2348), ADR(gc_DbmTranslation_en_Text2349), ADR(gc_DbmTranslation_en_Text2350), ADR(gc_DbmTranslation_en_Text2351), ADR(gc_DbmTranslation_en_Text2352), ADR(gc_DbmTranslation_en_Text2353), ADR(gc_DbmTranslation_en_Text2354), ADR(gc_DbVarGrpNameTranslation_en_Text2355), ADR(gc_DbVarGrpNameTranslation_en_Text2356), ADR(gc_DbVarGrpNameTranslation_en_Text2357), ADR(gc_DbVarGrpNameTranslation_en_Text2358), ADR(gc_DbVarGrpNameTranslation_en_Text2359), ADR(gc_DbVarGrpNameTranslation_en_Text2360), ADR(gc_DbVarGrpNameTranslation_en_Text2361), ADR(gc_DbVarGrpNameTranslation_en_Text2362), ADR(gc_DbVarGrpNameTranslation_en_Text2363), ADR(gc_DbVarGrpNameTranslation_en_Text2364), ADR(gc_DbVarGrpNameTranslation_en_Text2365), ADR(gc_DbVarGrpNameTranslation_en_Text2366), ADR(gc_DbVarGrpNameTranslation_en_Text2367), ADR(gc_DbVarGrpNameTranslation_en_Text2368), ADR(gc_DbVarGrpNameTranslation_en_Text2369), ADR(gc_DbVarGrpNameTranslation_en_Text2370), ADR(gc_DbVarGrpNameTranslation_en_Text2371)];
  gc_DbmTranslation_en : TTranslation := (IsoCode := 'en', EnglishName := "english", NativeName := "english", Texts := ADR(gc_DbmTranslation_en_Texts));
  gc_DbmTranslation_fr_Text0 : WSTRING(39) := "Pressure Block Oscillation Sensor State";
  gc_DbmTranslation_fr_Text1 : WSTRING(39) := "Pressure Block Oscillation Sensor Value";
  gc_DbmTranslation_fr_Text2 : WSTRING(43) := "Pressure Block Oscillation Sensor Raw value";
  gc_DbmTranslation_fr_Text3 : WSTRING(27) := "Pressure Brake Sensor State";
  gc_DbmTranslation_fr_Text4 : WSTRING(27) := "Pressure Brake Sensor Value";
  gc_DbmTranslation_fr_Text5 : WSTRING(31) := "Pressure Brake Sensor Raw value";
  gc_DbmTranslation_fr_Text6 : WSTRING(37) := "Temperature Transmission Sensor State";
  gc_DbmTranslation_fr_Text7 : WSTRING(37) := "Temperature Transmission Sensor Value";
  gc_DbmTranslation_fr_Text8 : WSTRING(41) := "Temperature Transmission Sensor Raw value";
  gc_DbmTranslation_fr_Text9 : WSTRING(25) := "Fault Pvg Left Trak State";
  gc_DbmTranslation_fr_Text10 : WSTRING(29) := "Fault Pvg Left Trak Raw Value";
  gc_DbmTranslation_fr_Text11 : WSTRING(26) := "Fault Pvg Right Trak State";
  gc_DbmTranslation_fr_Text12 : WSTRING(30) := "Fault Pvg Right Trak Raw value";
  gc_DbmTranslation_fr_Text13 : WSTRING(25) := "Down Axle oscillant State";
  gc_DbmTranslation_fr_Text14 : WSTRING(39) := "Down Axle oscillant  Raw value pin 0 Nc";
  gc_DbmTranslation_fr_Text15 : WSTRING(39) := "Down Axle oscillant  Raw value pin 1 No";
  gc_DbmTranslation_fr_Text16 : WSTRING(20) := "Down Axle fixe state";
  gc_DbmTranslation_fr_Text17 : WSTRING(24) := "Down Axle fixe Raw value";
  gc_DbmTranslation_fr_Text18 : WSTRING(33) := "Down Axle fixe Raw value pin 1 No";
  gc_DbmTranslation_fr_Text19 : WSTRING(23) := "Up Axle oscillant state";
  gc_DbmTranslation_fr_Text20 : WSTRING(23) := "Up Axle oscillant value";
  gc_DbmTranslation_fr_Text21 : WSTRING(18) := "Up Axle fixe state";
  gc_DbmTranslation_fr_Text22 : WSTRING(22) := "Up Axle fixe raw value";
  gc_DbmTranslation_fr_Text23 : WSTRING(29) := "Frame rotation sensor 1 state";
  gc_DbmTranslation_fr_Text24 : WSTRING(33) := "Frame rotation sensor 1 raw value";
  gc_DbmTranslation_fr_Text25 : WSTRING(39) := "Frame rotation sensor 1 raw value Pin 1";
  gc_DbmTranslation_fr_Text26 : WSTRING(22) := "Rail hook sensor state";
  gc_DbmTranslation_fr_Text27 : WSTRING(26) := "Rail hook sensor raw value";
  gc_DbmTranslation_fr_Text28 : WSTRING(27) := "Inductive Rail sensor state";
  gc_DbmTranslation_fr_Text29 : WSTRING(31) := "Inductive Rail sensor raw value";
  gc_DbmTranslation_fr_Text30 : WSTRING(21) := "Centered turret state";
  gc_DbmTranslation_fr_Text31 : WSTRING(25) := "Centered turret raw value";
  gc_DbmTranslation_fr_Text32 : WSTRING(25) := "Work Key track Side state";
  gc_DbmTranslation_fr_Text33 : WSTRING(29) := "Work Key track Side raw value";
  gc_DbmTranslation_fr_Text34 : WSTRING(29) := "Frame rotation sensor 2 state";
  gc_DbmTranslation_fr_Text35 : WSTRING(39) := "Frame rotation sensor 2 raw value Pin 0";
  gc_DbmTranslation_fr_Text36 : WSTRING(39) := "Frame rotation sensor 2 raw value Pin 1";
  gc_DbmTranslation_fr_Text37 : WSTRING(24) := "Work Key Bilateral state";
  gc_DbmTranslation_fr_Text38 : WSTRING(28) := "Work Key Bilateral raw value";
  gc_DbmTranslation_fr_Text39 : WSTRING(22) := "Work Key Centred state";
  gc_DbmTranslation_fr_Text40 : WSTRING(26) := "Work Key Centred raw value";
  gc_DbmTranslation_fr_Text41 : WSTRING(32) := "Abutment turret track side state";
  gc_DbmTranslation_fr_Text42 : WSTRING(36) := "Abutment turret track side raw value";
  gc_DbmTranslation_fr_Text43 : WSTRING(34) := "Abutment Turret Centred Side state";
  gc_DbmTranslation_fr_Text44 : WSTRING(38) := "Abutment Turret Centred Side raw value";
  gc_DbmTranslation_fr_Text45 : WSTRING(43) := "Oscillant Axle Speed Sensor Direction state";
  gc_DbmTranslation_fr_Text46 : WSTRING(47) := "Oscillant Axle Speed Sensor Direction Raw value";
  gc_DbmTranslation_fr_Text47 : WSTRING(38) := "Fixe Axle Speed Sensor Direction state";
  gc_DbmTranslation_fr_Text48 : WSTRING(42) := "Fixe Axle Speed Sensor Direction Raw value";
  gc_DbmTranslation_fr_Text49 : WSTRING(19) := "Trailer gache state";
  gc_DbmTranslation_fr_Text50 : WSTRING(23) := "Trailer gache raw value";
  gc_DbmTranslation_fr_Text51 : WSTRING(34) := "Measuring mast sensor folded state";
  gc_DbmTranslation_fr_Text52 : WSTRING(38) := "Measuring mast sensor folded raw value";
  gc_DbmTranslation_fr_Text53 : WSTRING(24) := "Oscillant Axle frequency";
  gc_DbmTranslation_fr_Text54 : WSTRING(19) := "Fixe Axle frequency";
  gc_DbmTranslation_fr_Text55 : WSTRING(25) := "Aru Radio 1 Contact state";
  gc_DbmTranslation_fr_Text56 : WSTRING(29) := "Aru Radio 1 Contact raw value";
  gc_DbmTranslation_fr_Text57 : WSTRING(25) := "Aru Radio 2 Contact state";
  gc_DbmTranslation_fr_Text58 : WSTRING(29) := "Aru Radio 2 Contact raw value";
  gc_DbmTranslation_fr_Text59 : WSTRING(19) := "Aru 1 Contact state";
  gc_DbmTranslation_fr_Text60 : WSTRING(23) := "Aru 1 Contact raw value";
  gc_DbmTranslation_fr_Text61 : WSTRING(19) := "Aru 2 Contact state";
  gc_DbmTranslation_fr_Text62 : WSTRING(23) := "Aru 2 contact raw value";
  gc_DbmTranslation_fr_Text63 : WSTRING(19) := "Starter motor state";
  gc_DbmTranslation_fr_Text64 : WSTRING(23) := "Starter motor raw value";
  gc_DbmTranslation_fr_Text65 : WSTRING(33) := "Autorisation High Speed Key State";
  gc_DbmTranslation_fr_Text66 : WSTRING(37) := "Autorisation High Speed Key Raw Value";
  gc_DbmTranslation_fr_Text67 : WSTRING(35) := "Electric pump Pressure Sensor State";
  gc_DbmTranslation_fr_Text68 : WSTRING(35) := "Electric pump Pressure Sensor Value";
  gc_DbmTranslation_fr_Text69 : WSTRING(39) := "Electric pump Pressure Sensor Raw value";
  gc_DbmTranslation_fr_Text70 : WSTRING(29) := "Mast sensor position UP State";
  gc_DbmTranslation_fr_Text71 : WSTRING(33) := "Mast sensor position UP Raw Value";
  gc_DbmTranslation_fr_Text72 : WSTRING(46) := "Hydraulic valve uin down position sensor state";
  gc_DbmTranslation_fr_Text73 : WSTRING(50) := "Hydraulic valve uin down position sensor raw value";
  gc_DbmTranslation_fr_Text74 : WSTRING(33) := "Ev Deflector Transmission command";
  gc_DbmTranslation_fr_Text75 : WSTRING(38) := "Ev Deflector Transmission actual value";
  gc_DbmTranslation_fr_Text76 : WSTRING(28) := "Ev Up Measuring Mast command";
  gc_DbmTranslation_fr_Text77 : WSTRING(33) := "Ev Up Measuring Mast actual value";
  gc_DbmTranslation_fr_Text78 : WSTRING(30) := "Ev Down Measuring Mast command";
  gc_DbmTranslation_fr_Text79 : WSTRING(35) := "Ev Down Measuring Mast actual value";
  gc_DbmTranslation_fr_Text80 : WSTRING(30) := "Ev Service Brake Track command";
  gc_DbmTranslation_fr_Text81 : WSTRING(35) := "Ev Service Brake Track actual value";
  gc_DbmTranslation_fr_Text82 : WSTRING(26) := "Ev Power Reduction command";
  gc_DbmTranslation_fr_Text83 : WSTRING(31) := "Ev Power Reduction actual value";
  gc_DbmTranslation_fr_Text84 : WSTRING(27) := "Ev Frame Rotation 1 command";
  gc_DbmTranslation_fr_Text85 : WSTRING(32) := "Ev Frame Rotation 1 actual value";
  gc_DbmTranslation_fr_Text86 : WSTRING(27) := "Ev Frame Rotation 2 command";
  gc_DbmTranslation_fr_Text87 : WSTRING(32) := "Ev Frame Rotation 2 actual value";
  gc_DbmTranslation_fr_Text88 : WSTRING(29) := "Supply Radio Receiver command";
  gc_DbmTranslation_fr_Text89 : WSTRING(34) := "Supply Radio Receiver actual value";
  gc_DbmTranslation_fr_Text90 : WSTRING(34) := "Buzzer Lynx Moving Machine command";
  gc_DbmTranslation_fr_Text91 : WSTRING(39) := "Buzzer Lynx Moving Machine actual value";
  gc_DbmTranslation_fr_Text92 : WSTRING(28) := "White Lights Trailer command";
  gc_DbmTranslation_fr_Text93 : WSTRING(33) := "White Lights Trailer actual value";
  gc_DbmTranslation_fr_Text94 : WSTRING(26) := "Red Lights Trailer command";
  gc_DbmTranslation_fr_Text95 : WSTRING(31) := "Red Lights Trailer actual value";
  gc_DbmTranslation_fr_Text96 : WSTRING(23) := "White Light AVG command";
